// TIA Portal V18 program export: 3 tag tables, 18 data types, 3 data blocks, 44 code blocks (in call order from the OBs), 34 instance data blocks

VAR_GLOBAL   // PLC tag table "Assigned IO"
   HPU_In AT %I0.0 : "Starter_HPU_IO_In";
   HPU_Out AT %Q0.0 : "Starter_HPU_IO_Out";
   Console_In AT %I200.0 : "Console_IO_In";
   Console_Out AT %Q200.0 : "Console_IO_Out";
   ComFault AT %M20.1 : Bool;
   SystemFault AT %M1.0 : Bool;
   RemConsole_In AT %I500.0 : "RemConsole_IO_In";
   RemConsole_Out AT %Q500.0 : "RemConsole_IO_Out";
   RemConEn AT %M29.6 : Bool;   // Remote console is enable if Aux or TD En and heartbeat is ok
END_VAR

VAR_GLOBAL   // PLC tag table "Default tag table"
   TestByte AT %MB2500 : Byte;
   RotaryRPMHMI AT %MD534 : Real;   // It is a absolute value, to display on HMI gauge
   PSIcheck AT %MD544 : Real;
   RotaryStopped AT %M568.0 : Bool;
   MUTorqSetKFtLbs AT %MD570 : Real;
   DrillTorqSetKFtLbs AT %MD574 : Real;
END_VAR
VAR_GLOBAL CONSTANT   // user constants
   RigNumber : Real := 0.0;
   "Program Version" : Real := 0.0;
   RotaryEncInvDir : Bool := 0;   // Used to invert the counting of the rotary encoder
END_VAR

VAR_GLOBAL   // PLC tag table "System Variables"
   RotaryCounts AT %MD100 : DInt;   // Actually rotary count feedback
   RotaryRPM AT %MD104 : Real;   // frequency of rotray feedack
   AuxPumpRunning AT %M10.0 : Bool;   // Status of Aux Pump. 1 Running 0 stopped
   EngineRPMCounts AT %MD108 : DInt;   // CAT Engine RPM count return
   EngineRPMFreq AT %MD112 : Real;   // CAT Engine RPM freqency measured
   CoolingFanRunning AT %M10.1 : Bool;   // Status of Cooler Running 0 stopped
   M1Running AT %M10.2 : Bool;   // Status of P1 Running 0 stopped
   M2Running AT %M10.3 : Bool;   // Status of P2 Running 0 stopped
   AuxPumpHOA AT %M10.4 : Bool;   // Actual Signal to Soft Starter
   CoolingFanHOA AT %M10.5 : Bool;   // Actual Signal to Soft Starter
   M1HOA AT %M10.6 : Bool;   // Actual Signal to Soft Starter
   M2HOA AT %M10.7 : Bool;   // Actual Signal to Soft Starter
   ChargePump1PSw AT %M11.0 : Bool;   // Close = Pressure
   TDLubeFlowSw AT %M11.1 : Bool;   // Close = Flow
   TankLowLevelSw AT %M11.2 : Bool;   // Low Level = Open
   TankHighTempSw AT %M11.3 : Bool;   // High Temp = Open
   TDFwdFilter2 AT %M11.5 : Bool;   // Plugged = Open
   TDRevFilter1 AT %M11.6 : Bool;   // Plugged = Open
   TDRevFilter2 AT %M11.7 : Bool;   // Plugged = Open
   AuxReturnFilter AT %M12.0 : Bool;   // Plugged = Open
   KLoopFilter AT %M12.1 : Bool;   // Plugged = Open
   ChargeFilter AT %M12.2 : Bool;   // Plugged = Open
   M1CurrentRaw AT %MW122 : Int;
   M2CurrentRaw AT %MW128 : Int;
   M1CurrentV AT %MD124 : Real;
   M2CurrentV AT %MD130 : Real;
   TDPressFWDRaw AT %MW134 : Int;   // TD Forward Pressure Input
   TDPressREVRaw AT %MW136 : Int;   // TD Reverse Pressure Input
   ClosedLoopTempRaw AT %MW138 : Int;
   ChargeFlowRaw AT %MW140 : Int;
   HotOilShuttleFlowRaw AT %MW142 : Int;
   AuxFlowRaw AT %MW144 : Int;
   ChargePress1Raw AT %MW146 : Int;
   ChargePress2Raw AT %MW148 : Int;
   TDPressFWDmA AT %MD150 : Real;   // TD Forward Pressure Input
   TDPressREVmA AT %MD154 : Real;   // TD Reverse Pressure Input
   ClosedLoopTempmA AT %MD158 : Real;
   ChargeFlowmA AT %MD162 : Real;
   HotOilShuttleFlowmA AT %MD166 : Real;
   AuxFlowmA AT %MD170 : Real;
   ChargePress1mA AT %MD174 : Real;
   ChargePress2mA AT %MD178 : Real;
   TDP1FwdCmdActRaw AT %MW182 : Int;   // Actual measured output to valve from module
   TDP1RevCmdActRaw AT %MW184 : Int;   // Actual measured output to valve from module
   TDP2FwdCmdActRaw AT %MW186 : Int;   // Actual measured output to valve from module
   TDP2RevCmdActRaw AT %MW188 : Int;   // Actual measured output to valve from module
   TDTorqCmdActRaw AT %MW190 : Int;   // Raw Output to card
   TDP1FwdCmdActmA AT %MD192 : Real;   // Actual measured output to valve from module
   TDP1RevCmdActmA AT %MD196 : Real;   // Actual measured output to valve from module
   TDP2FwdCmdActmA AT %MD200 : Real;   // Actual measured output to valve from module
   TDP2RevCmdActmA AT %MD204 : Real;   // Actual measured output to valve from module
   TDTorqCmdActmA AT %MD208 : Real;   // Actual measured output to valve from module
   LinkRetSw AT %M12.4 : Bool;   // Console Input
   TDAuxSw AT %M12.5 : Bool;   // Console Input
   LinkExtSw AT %M12.6 : Bool;   // Console Input
   TDEnSW AT %M12.7 : Bool;   // Console Input
   HSLT_Sw AT %M13.0 : Bool;   // Console Input
   HandlerFwdSw AT %M13.1 : Bool;   // Console Input
   HandlerRevSw AT %M13.2 : Bool;   // Console Input
   MPNotRunning AT %M13.3 : Bool;   // 0 Pump Running, 1 Pump Not Running - Allowed to Run. Power to permit
   QuillLockSw AT %M13.4 : Bool;   // Console Input
   BUWClSw AT %M13.5 : Bool;   // Console Input
   BUWDnSw AT %M13.6 : Bool;   // Console Input
   BUWUpSw AT %M13.7 : Bool;   // Console Input
   TDModeMUSpinSw AT %M14.0 : Bool;   // Console Input
   TDModeMUTorqSw AT %M14.1 : Bool;   // Console Input
   TDModeDrillRevSw AT %M14.2 : Bool;   // Console Input
   TDModeBreakOutSw AT %M14.3 : Bool;   // Console Input
   ElevOpSw AT %M14.4 : Bool;   // Console Input
   TDExtSw AT %M14.5 : Bool;   // Console Input
   ElevClSw AT %M14.6 : Bool;   // Console Input
   TDRetSw AT %M14.7 : Bool;   // Console Input
   PTO_Sw AT %M15.0 : Bool;   // Console Input
   PurgePressureSw AT %M15.1 : Bool;   // Console Input
   MSVClSw AT %M15.2 : Bool;   // Console Input
   MSVAutoSw AT %M15.3 : Bool;   // Console Input
   MSVOpSw AT %M15.4 : Bool;   // Console Input
   LinkFloatSw AT %M15.5 : Bool;   // Console Input
   MUTorqPotRaw AT %MW212 : Int;
   DrillTorqPotRaw AT %MW214 : Int;
   DrillThrottlePotRaw AT %MW216 : Int;
   MUTorqPotV AT %MD218 : Real;
   DrillTorqPotV AT %MD222 : Real;
   DrillThrottlePotV AT %MD226 : Real;
   RotEncLDSlot AT %MB230 : Byte;   // Bit 0-3 Slot 0, Bit 4-7 Slot 1. 0 0 0 0 for Idle, 0 0 0 1 Load Counter
   TDFwdPress1Raw AT %MD240 : UDInt;   // Pump 1 Forward Pressure output
   TDFwdPress2Raw AT %MD244 : UDInt;   // Pump 2 Forward Pressure output
   TDRevPress1Raw AT %MD248 : UDInt;   // Pump 1 Rev Pressure output
   TDRevPress2Raw AT %MD252 : UDInt;   // Pump 2 Rev Pressure output
   TDTorqPressRaw AT %MD256 : UDInt;   // Torq Output
   TDFwdPress1En AT %M15.6 : Bool;   // Enable Pump 1 Forward Pressure output
   TDFwdPress2En AT %M15.7 : Bool;   // Enable Pump 2 Forward Pressure output
   TDRevPress1En AT %M16.0 : Bool;   // Enable Pump 1 Rev Pressure output
   TDRevPress2En AT %M16.1 : Bool;   // Enable Pump 2 Rev Pressure output
   TDTorqPressEn AT %M16.2 : Bool;   // Enable Torq output
   BUWClSol AT %M16.4 : Bool;
   HSLT_Sol AT %M16.5 : Bool;
   ElevClSol AT %M16.6 : Bool;
   ElevOpSol AT %M16.7 : Bool;
   LinkExtSol AT %M17.0 : Bool;
   LinkRetSol AT %M17.1 : Bool;
   LinkFloatSol AT %M17.2 : Bool;
   LSHT_Sol AT %M17.3 : Bool;
   MSVOpSol AT %M17.4 : Bool;
   MSVClSol AT %M17.5 : Bool;
   BUWDnSol AT %M17.6 : Bool;
   BUWUpSol AT %M17.7 : Bool;
   HandlerFWDSol AT %M18.0 : Bool;
   HandlerREVSol AT %M18.1 : Bool;
   TDExtSol AT %M18.2 : Bool;
   TDRetSol AT %M18.3 : Bool;   // Output Coil
   HourMeterOn AT %M18.4 : Bool;
   EngRampSpeedDn AT %M18.5 : Bool;
   AuxPumpStart AT %M18.6 : Bool;
   EngRampSpeedUp AT %M18.7 : Bool;
   CoolingFanStart AT %M19.0 : Bool;
   FailSafeEnSol AT %M19.1 : Bool;
   PumpEnSol AT %M19.2 : Bool;   // CAT/Rig 11 Only
   BOControlSol AT %M19.3 : Bool;
   AuxUnloaderSol AT %M19.4 : Bool;
   HotOilControlSol AT %M19.5 : Bool;
   BUWOpSol AT %M19.6 : Bool;
   BypassValveSol AT %M19.7 : Bool;
   TDFwdPress1mA AT %MD260 : Real;   // Pump 1 Forward Pressure output
   TDFwdPress2mA AT %MD264 : Real;   // Pump 2 Forward Pressure output
   TDRevPress1mA AT %MD268 : Real;   // Pump 1 Rev Pressure output
   TDRevPress2mA AT %MD272 : Real;   // Pump 2 Rev Pressure output
   TDTorqPressmA AT %MD276 : Real;   // Torq Output
   PTOLED AT %M20.4 : Bool;
   HPUFaultLED AT %M20.5 : Bool;
   TDFlushFaultLED AT %M20.6 : Bool;
   BUWClLED AT %M20.7 : Bool;
   TDEnLED AT %M21.0 : Bool;
   ConLowPurgeLED AT %M21.1 : Bool;
   MSVClLED AT %M21.2 : Bool;   // Mud Saver valve closed LED
   QuillLockLED AT %M21.3 : Bool;
   ElevClLED AT %M21.4 : Bool;
   Horn AT %M21.5 : Bool;
   MSVClInt AT %M21.6 : Bool;   // Mud saver valve closed interlocks outputs
   BUWClInt AT %M21.7 : Bool;   // BUW Closed interlock outputs
   DrillRecTorqRaw AT %MW280 : Int;
   DrillRecRPMRaw AT %MW282 : Int;
   DrillRecTorqFtLbs AT %MD284 : Real;
   DrillRecRPM AT %MD288 : Real;
   DrillRecTorqmA AT %MD292 : Real;
   DrillRecRPMmA AT %MD296 : Real;
   RotEncUnFl AT %M22.0 : Bool;   // Encoder underflow
   RotEncOvFl AT %M22.1 : Bool;   // Encoder OVerflow
   RotEncPosReset AT %M22.2 : Bool;   // Set high to trigger zero position of encoder. Bit will reset once position reset
   RotEncSlot0 AT %MD232 : Real;
   RotEncSlot1 AT %MD236 : Real;
   TDRotStopped AT %M22.3 : Bool;   // Set if TD has not moved after stop time elapsed
   RotAbsPosDeg AT %MD300 : Real;   // Absolute rotary position from zero point
   RotRelPosDeg AT %MD304 : Real;   // Position from 0-360 degrees
   RotPosTurns AT %MD308 : Real;   // Turns from zero point
   TDFlushFlowSw AT %M22.4 : Bool;
   M1Current AT %MD312 : Real;
   M2Current AT %MD316 : Real;
   TDPressFwdPSI AT %MD320 : Real;   // TD Fwd Pressure PSI
   TDPressRevPSI AT %MD324 : Real;   // TD Rev Pressure PSI
   ClosedLoopTempC AT %MD328 : Real;   // Closed Loop Temp in C
   ChargeFlowGPM AT %MD332 : Real;   // Charge Flow in GPM
   HotOilFlowGPM AT %MD336 : Real;   // Hot Oil Shuttle Flow in GPM
   AuxFlowGPM AT %MD340 : Real;   // Aux Flow GPM
   ChargePress1PSI AT %MD344 : Real;   // Charge Pump 1 Pressure PSI
   ChargePress2PSI AT %MD348 : Real;   // Charge Pump 2 Pressure PSI
   M1CurrentFilt AT %MD352 : Real;
   M2CurrentFilt AT %MD356 : Real;
   TDPressFwdPSIFilt AT %MD360 : Real;
   TDPressRevPSIFilt AT %MD364 : Real;
   ClosedLoopTempCFilt AT %MD368 : Real;
   ChargeFlowGPMFilt AT %MD372 : Real;
   HotOilFlowGPMFilt AT %MD376 : Real;
   AuxFlowGPMFilt AT %MD380 : Real;
   ChargePress1PSIFilt AT %MD384 : Real;
   ChargePress2PSIFilt AT %MD388 : Real;
   AuxPumpHand AT %M22.5 : Bool;   // Starter HOA switch in the Hand Position
   AuxPumpOff AT %M22.6 : Bool;   // Starter HOA switch in the Off position
   CoolingFanHand AT %M23.0 : Bool;   // Starter HOA switch in the Hand Position
   CoolingFanOff AT %M23.1 : Bool;   // Starter HOA switch in the Off position
   M1Hand AT %M23.3 : Bool;   // Starter HOA switch in the Hand Position
   M1Off AT %M23.4 : Bool;   // Starter HOA switch in the Off position
   M2Hand AT %M23.6 : Bool;   // Starter HOA switch in the Hand Position
   M2Off AT %M23.7 : Bool;   // Starter HOA switch in the Off position
   AuxPumpFault AT %M22.7 : Bool;   // Motor failed to start before motor timeout time
   CoolingFanFault AT %M23.2 : Bool;   // Motor failed to start before motor timeout time
   M1Fault AT %M23.5 : Bool;   // Motor failed to start before motor timeout time
   M2Fault AT %M24.0 : Bool;   // Motor failed to start before motor timeout time
   M1Start AT %M20.2 : Bool;   // Start Motor 1
   M2Start AT %M20.3 : Bool;   // Start Motor 2
   BypassStart AT %M24.1 : Bool;   // Ready for Bypass to start, waiting for PTO
   BypassRunning AT %M24.2 : Bool;   // Latched Signal set if PTO pressed after Bypass Start
   StartCAT AT %M24.3 : Bool;   // Indicates CAT startup up. System ramps up and will enable.
   BUWMaintConfirm AT %M24.4 : Bool;
   PTOConfirmed AT %M24.5 : Bool;   // PTO Confirm pulse for 5 seconds after button pressed
   BUWOpenClk AT %M24.6 : Bool;   // Periodic clock signal that will be on for 5 seconds and off for 1 min. Used for maintain gripper open
   BUWAutoCl AT %M24.7 : Bool;   // Latch for Gripper Close
   BUWAutoClHold AT %M25.0 : Bool;   // LAtch for Gripper Hold Closed
   BUWAutoOp AT %M25.1 : Bool;   // Lath for Gripper Open
   OscSpeedfwdHold AT %M25.2 : Bool;
   QuillLockEnabled AT %M25.3 : Bool;   // Bit used to know if Quill Lock allowed
   BUWClHoldTime AT %M25.4 : Bool;   // On for half a second to hold the close before turning off
   MUTorqPotPer AT %MD392 : Real;
   DrillTorqPotPer AT %MD396 : Real;
   DrillThrottlePotPer AT %MD400 : Real;
   MUTorqPotPerFilt AT %MD404 : Real;
   DrillTorqPotPerFilt AT %MD408 : Real;
   DrillThrottlePotPerFilt AT %MD412 : Real;
   ActTorqFtLbs AT %MD416 : Real;   // Calculated actual torque
   ActTorqFtLbsFilt AT %MD420 : Real;   // Filtered Actual Torque
   TDDifPressPSI AT %MD424 : Real;   // Diffential pressure betweeen FWD and REV
   DrillTorqSetFtLbs AT %MD428 : Real;   // Internal setpoint value from the console input FtLbs
   MUTorqSetFtLbs AT %MD432 : Real;   // Internal setpoint value from the console input FtLbs
   RotDegPerCount AT %MD436 : Real;   // Actual Degrees per Count for current encoder setup
   DrillTorqSetMax AT %MD440 : Real;   // Maximum value allowed to set drill torq too based on MU torq settings
   BOCycleDone AT %M25.6 : Bool;   // Trigger when BO Sw released
   MUCycleDone AT %M25.7 : Bool;   // Set when MU done
   MUSwRelease AT %M26.0 : Bool;   // Trigger when MU SW released
   MUDoneSetFtLbs AT %MD444 : Real;   // Minimum torque to surpass to declare MU Done
   ElevClFeedback AT %M12.3 : Bool;   // Feedback switch that the elevators are closed
   LamptTest AT %M26.1 : Bool;   // Bit Used to trigger Lamp to turn on.
   FlushFaultNoSpin AT %M26.2 : Bool;   // TD flush faulted. No Spin allowed
   ThrottleDisable AT %M26.3 : Bool;   // Throttle disable if high
   ThrottleUnlocked AT %M26.4 : Bool;   // Throttle boots up locked. Must be below zero to enable after startup
   DrillTorqLimited AT %M26.5 : Bool;   // Set high if max drill torq limited by max makeup torq
   DrillTorqSetPSI AT %MD448 : Real;   // PSI equivalent to get desired torq from valve
   MUTorqSetPSI AT %MD452 : Real;   // PSI equivalent to get desired torq from valve
   TDStart AT %M25.5 : Bool;   // Bit will be set High when TD is started for regular operations
   BypassPTO AT %M26.6 : Bool;   // Bypass PTO accept
   BypassOutEnable AT %M26.7 : Bool;   // Bypass control enabled to allow signal to Pumps after delay
   BypassHighTemp AT %M27.0 : Bool;   // High Closed loop temp in bypass mode
   TDPressTxFault AT %M27.1 : Bool;   // One of the pressure transducers if not working. No auto MU
   HSLTDisThrottle AT %M27.2 : Bool;   // Bit high after shift to disable throttle
   LSHTDisThrottle AT %M27.3 : Bool;   // Bit high after shift to disable throttle
   MUSeqRunning AT %M27.4 : Bool;   // Bool indicating mak up sequence is running.
   AutoMUTorqLow AT %M27.5 : Bool;   // Auto Make Up Low Torque range
   AutoMUTorqMid AT %M27.6 : Bool;   // Auto Make Up Mid Torque Range
   AutoMuTorqHigh AT %M27.7 : Bool;   // Auto Make Up High Torque Range
   HiTempRPMRed AT %M28.1 : Bool;   // Bit indicating high temperature and RPM to be reduced
   HiTempShutdown AT %M28.2 : Bool;   // Bit indicating high temperature and shutdown needed.
   TDRotDirFwd AT %M28.3 : Bool;   // Rotary moving fwd
   TDRotDirRev AT %M28.4 : Bool;   // Rotary moving rev
   ActTorqKFtLbsFilt AT %MD456 : Real;
   RotEncA AT %M28.5 : Bool;
   RotEncB AT %M28.6 : Bool;
   BOSeqRunning AT %M28.0 : Bool;   // Bool indicating break out sequence is running.   {ExternalVisible false}
   HPU_AiV2SpareRaw AT %MW460 : Int;   // Spare Analog Voltage Input Raw
   HPU_AiV2SpareV AT %MD472 : Real;   // Spare Analog Voltage Input
   HPU_AiV3SpareRaw AT %MW462 : Int;   // Spare Analog Voltage Input Raw
   HPU_AiV4SpareRaw AT %MW464 : Int;   // Spare Analog Voltage Input Raw
   HPU_AiV5SpareRaw AT %MW466 : Int;   // Spare Analog Voltage Input Raw
   HPU_AiV6SpareRaw AT %MW468 : Int;   // Spare Analog Voltage Input Raw
   HPU_AiV7SpareRaw AT %MW470 : Int;   // Spare Analog Voltage Input Raw
   HPU_AiV3SpareV AT %MD476 : Real;   // Spare Analog Voltage Input
   HPU_AiV4SpareV AT %MD480 : Real;   // Spare Analog Voltage Input
   HPU_AiV5SpareV AT %MD484 : Real;   // Spare Analog Voltage Input
   HPU_AiV6SpareV AT %MD488 : Real;   // Spare Analog Voltage Input
   HPU_AiV7SpareV AT %MD492 : Real;   // Spare Analog Voltage Input
   Con_AiV3SpareRaw AT %MW496 : Int;   // Spare Analog Voltage Input Raw
   Con_AiV4SpareRaw AT %MW498 : Int;   // Spare Analog Voltage Input Raw
   Con_AiV5SpareRaw AT %MW500 : Int;   // Spare Analog Voltage Input Raw
   Con_AiV6SpareRaw AT %MW502 : Int;   // Spare Analog Voltage Input Raw
   Con_AiV7SpareRaw AT %MW504 : Int;   // Spare Analog Voltage Input Raw
   Con_AiV3SpareV AT %MD506 : Real;   // Spare Analog Voltage Input
   Con_AiV4SpareV AT %MD510 : Real;   // Spare Analog Voltage Input
   Con_AiV5SpareV AT %MD514 : Real;   // Spare Analog Voltage Input
   Con_AiV6SpareV AT %MD518 : Real;   // Spare Analog Voltage Input
   Con_AiV7SpareV AT %MD522 : Real;   // Spare Analog Voltage Input
   HornTest AT %M28.7 : Bool;
   Charge1Fault AT %M29.0 : Bool;   // Charge pressure fault while TD enabled
   FilterPlugged AT %M29.1 : Bool;
   Clock_Byte AT %MB0 : Byte;
   Clock_10Hz AT %M0.0 : Bool;   // 0.1 s period
   Clock_5Hz AT %M0.1 : Bool;   // 0.2 s period
   "Clock_2.5Hz" AT %M0.2 : Bool;   // 0.4 s period
   Clock_2Hz AT %M0.3 : Bool;   // .06 s period
   "Clock_1.25Hz" AT %M0.4 : Bool;   // 0.8s period
   Clock_1Hz AT %M0.5 : Bool;   // 1s period
   "Clock_0.625Hz" AT %M0.6 : Bool;   // 1.6s period
   "Clock_0.5Hz" AT %M0.7 : Bool;   // 2.0 s period
   HiTempAlarm AT %M29.2 : Bool;
   LubeFlowFault AT %M29.3 : Bool;
   HornSilence AT %M29.4 : Bool;
   EngineFault AT %M29.5 : Bool;   // CAT Engine Fault. Below min RPM
   EngineRPM AT %MD116 : Real;
   ClosedLoopTempCMax AT %MD526 : Real;
   TDEnabled AT %M16.3 : Bool;   // Start Request received and system enabled
   Charge2Fault AT %M20.0 : Bool;
   ChargePump2PSw AT %M29.7 : Bool;   // Close = Pressure
   TDFwdFilter1 AT %M11.4 : Bool;   // Plugged = Open
   LastCount AT %MD30 : DInt;
   RotRelPosDegHMIPos AT %MD34 : Real;
   OscHomeRelDegHMIPos AT %MD530 : Real;
   SwitchSWGATE AT %M538.0 : Bool;
   OscSpeedrevHold AT %M38.0 : Bool;
   RevFwdPause AT %M38.1 : Bool;
   FwdRevPasue AT %M38.2 : Bool;
   PSIadjustbit AT %M38.3 : Bool;
   PSIdrillTorquCalca AT %MD540 : Real;
   PSIsettle AT %MD548 : Real;
   PSIadjustRange AT %MD552 : Real;
   PSIadjustval AT %MD556 : Real;
   ClosedLoopTempF AT %MD560 : Real;
   RotaryRPMActual AT %MD564 : Real;
END_VAR
VAR_GLOBAL CONSTANT   // user constants
   AlwaysOn : Bool := 1;
   AlwaysOff : Bool := 0;
END_VAR

TYPE "Console_IO_In"
   STRUCT
      Slot1 { S7_SetPoint := 'True'} : "DI16x24V_In";
      Slot2 { S7_SetPoint := 'True'} : "DI16x24V_In";
      Slot3 { S7_SetPoint := 'True'} : "AI8xU_In";
   END_STRUCT;
END_TYPE

TYPE "Console_IO_Out"
   STRUCT
      Slot4 : "DQ16x24V_Out";
      Slot5 : "AQ4xI/U_Out";
   END_STRUCT;
END_TYPE

TYPE "RemConsole_IO_In"
   STRUCT
      Element_1 : Bool;
      Element_2 : Bool;
      Element_3 : Bool;
      Element_4 : Bool;
      Element_5 : Bool;
      Element_6 : Bool;
      Element_7 : Bool;
      LinkTiltRetr : Bool;
      TopDriveAux : Bool;
      LinkTiltExt : Bool;
      TopDriveEn : Bool;
      HSLTEn : Bool;
      HandlerFwd : Bool;
      HandlerRev : Bool;
      MudPumpRunning : Bool;
      QuillLock : Bool;
      BUWClose : Bool;
      BUWDown : Bool;
      BUWUp : Bool;
      TDModeMUSpin : Bool;
      TDModeMUTorq : Bool;
      TDModeRev : Bool;
      TDModeBO : Bool;
      ElevOp : Bool;
      TDExt : Bool;
      ElevCl : Bool;
      TDRet : Bool;
      PTO : Bool;
      Spare : Bool;
      MSVClose : Bool;
      MSVAuto : Bool;
      MSVOpen : Bool;
      LinkTiltFloat : Bool;
      Spare_1 : Bool;
      Spare_2 : Bool;
      Spare_3 : Bool;
      Spare_4 : Bool;
      Spare_5 : Bool;
      Heartbeat : Bool;
      Reserved : Byte;
      MUTorqLim : Int;
      DrillTorqLim : Int;
      DrillThrottle : Int;
      SpareAI : Int;
      SpareAI_1 : Int;
      SpareAI_2 : Int;
      SpareAI_3 : Int;
      SpareAI_1_1 : Int;
   END_STRUCT;
END_TYPE

TYPE "RemConsole_IO_Out"
   STRUCT
      PTOLED : Bool;
      HPUFaultLED : Bool;
      TDFaultLED : Bool;
      BUWClLED : Bool;
      TDEnLED : Bool;
      Spare_6 : Bool;
      MSVClLED : Bool;
      QuillLockedLED : Bool;
      ElevClLED : Bool;
      Horn : Bool;
      MSVClInt : Bool;
      BUWClInt : Bool;
      Spare_7 : Bool;
      Spare_8 : Bool;
      Spare_9 : Bool;
      Spare_10 : Bool;
      Spare_11 : Bool;
      Spare_12 : Bool;
      Spare_13 : Bool;
      Spare_14 : Bool;
      Spare_15 : Bool;
      Spare : Bool;
      Spare_16 : Bool;
      Spare_17 : Bool;
      Spare_18 : Bool;
      Spare_19 : Bool;
      Spare_1 : Bool;
      Spare_2 : Bool;
      Spare_3 : Bool;
      Spare_4 : Bool;
      Spare_5 : Bool;
      Spare_20 : Bool;
      DrillRecTorq : Int;
      DrillRecRPM : Int;
      SpareAO : Int;
      SpareAO_2 : Int;
   END_STRUCT;
END_TYPE

TYPE "Runtime_Out"
   STRUCT
      TotalTime : DInt;
      TotHours : DInt;
      TotMins : DInt;
      TotSeconds : DInt;
      CurrentTime : DInt;   // Current Time in Seconds
      CurHours : DInt;
      CurMins : DInt;
      CurSeconds : DInt;
   END_STRUCT;
END_TYPE

TYPE "Starter_HPU_IO_In"
   STRUCT
      Slot2 { ExternalWritable := 'False'} : "TM_Count_Man_In";
      Slot3 { ExternalWritable := 'False'} : "DI16x24V_In";
      Slot4 { ExternalWritable := 'False'} : "DI16x24V_In";
      Slot5 { S7_SetPoint := 'True'} : "AI8xU_In";
      Slot6 { ExternalWritable := 'False'} : "AI8xI_In";
      Slot7 { ExternalWritable := 'False'} : "TM_Pulse_2x24_In";
      Slot8 { S7_SetPoint := 'True'} : "TM_Pulse_2x24_In";
      Slot9 { S7_SetPoint := 'True'} : "TM_Pulse_2x24_In";
   END_STRUCT;
END_TYPE

TYPE "Starter_HPU_IO_Out"
   STRUCT
      Slot2 { S7_SetPoint := 'True'} : "TM_Count_Man_Out";
      Slot7 { S7_SetPoint := 'True'} : "TM_Pulse_2x24_Out";
      Slot8 { S7_SetPoint := 'True'} : "TM_Pulse_2x24_Out";
      Slot9 { S7_SetPoint := 'True'} : "TM_Pulse_2x24_Out";
      Slot10 { S7_SetPoint := 'True'} : "RQ_4x120VDC/5A_In";
      Slot11 { S7_SetPoint := 'True'} : "RQ_4x120VDC/5A_In";
      Slot12 { S7_SetPoint := 'True'} : "RQ_4x120VDC/5A_In";
      Slot13 { S7_SetPoint := 'True'} : "RQ_4x120VDC/5A_In";
      Slot14 { S7_SetPoint := 'True'} : "RQ_4x120VDC/5A_In";
      Slot15 { S7_SetPoint := 'True'} : "RQ_4x120VDC/5A_In";
      Slot16 { S7_SetPoint := 'True'} : "RQ_4x120VDC/5A_In";
      Slot17 { S7_SetPoint := 'True'} : "RQ_4x120VDC/5A_In";
   END_STRUCT;
END_TYPE

TYPE "TD_Modes"
   STRUCT
      Drill : Int;
      DrillReverse : Int := 1;
      MUSpin : Int := 2;
      MUTorque : Int := 3;
      BO : Int := 4;
      Oscillate : Int := 5;
      Bypass : Int := 6;
   END_STRUCT;
END_TYPE

TYPE "AI8xI_In"
   STRUCT
      Ch0 : Int;
      Ch1 : Int;
      Ch2 : Int;
      Ch3 : Int;
      Ch4 : Int;
      Ch5 : Int;
      Ch6 : Int;
      Ch7 : Int;
   END_STRUCT;
END_TYPE

TYPE "AI8xU_In"
   STRUCT
      Ch0 : Int;
      Ch1 : Int;
      Ch2 : Int;
      Ch3 : Int;
      Ch4 : Int;
      Ch5 : Int;
      Ch6 : Int;
      Ch7 : Int;
   END_STRUCT;
END_TYPE

TYPE "DI16x24V_In"
   STRUCT
      Ch0 : Bool;
      Ch1 : Bool;
      Ch2 : Bool;
      Ch3 : Bool;
      Ch4 : Bool;
      Ch5 : Bool;
      Ch6 : Bool;
      Ch7 : Bool;
      Ch8 : Bool;
      Ch9 : Bool;
      Ch10 : Bool;
      Ch11 : Bool;
      Ch12 : Bool;
      Ch13 : Bool;
      Ch14 : Bool;
      Ch15 : Bool;
   END_STRUCT;
END_TYPE

TYPE "DQ16x24V_Out"
   STRUCT
      Ch0 : Bool;
      Ch1 : Bool;
      Ch2 : Bool;
      Ch3 : Bool;
      Ch4 : Bool;
      Ch5 : Bool;
      Ch6 : Bool;
      Ch7 : Bool;
      Ch8 : Bool;
      Ch9 : Bool;
      Ch10 : Bool;
      Ch11 : Bool;
      Ch12 : Bool;
      Ch13 : Bool;
      Ch14 : Bool;
      Ch15 : Bool;
   END_STRUCT;
END_TYPE

TYPE "TM_Count_Man_In"
   STRUCT
      COUNT_VALUE : DInt;
      CAPTURED_VALUE : DInt;
      MEASURED_VALUE : DInt;
      POWER_ERROR : Bool;
      ENC_ERROR : Bool;
      LD_ERROR : Bool;
      Reserved1 : Bool;
      Reserved2 : Bool;
      Reserved3 : Bool;
      Reserved4 : Bool;
      Reserved5 : Bool;
      Reserved6 : Bool;
      RES_EVENT_ACK : Bool;
      LD_STS_SLOT0 : Bool;
      LD_STS_SLOT1 : Bool;
      STS_READY : Bool;
      STS_SW_GATE : Bool;
      Reserved7 : Bool;
      Reserved8 : Bool;
      STS_DIR : Bool;
      STS_CNT : Bool;
      STS_GATE : Bool;
      STS_DQ0 : Bool;
      STS_DQ1 : Bool;
      STS_DI0 : Bool;
      STS_DI1 : Bool;
      STS_DI2 : Bool;
      EVENT_ZERO : Bool;
      EVENT_UFLW : Bool;
      EVENT_OFLW : Bool;
      EVENT_CMP0 : Bool;
      EVENT_CMP1 : Bool;
      EVENT_SYNC : Bool;
      EVENT_CAP : Bool;
      STS_M_INTERVAL : Bool;
   END_STRUCT;
END_TYPE

TYPE "TM_Count_Man_Out"
   STRUCT
      SLOT_0 : Real;
      SLOT_1 : Real;
      LD_SLOT_0_1 : Byte;
      SW_GATE : Bool;
      TM_CTRL_DQ0 : Bool;
      TM_CTRL_DQ1 : Bool;
      SET_DQ0 : Bool;
      SET_DQ1 : Bool;
      EN_SYNC_UP : Bool;
      EN_SYNC_DN : Bool;
      EN_CAPTURE : Bool;
      RES_ERROR : Bool;
      RES_EVENT : Bool;
      Reserved1 : Bool;
      Reserved2 : Bool;
      Reserved3 : Bool;
      Reserved4 : Bool;
      Reserved5 : Bool;
      SET_DIR : Bool;
      Reserved : Byte;
   END_STRUCT;
END_TYPE

TYPE "TM_Pulse_2x24_In"
   STRUCT
      Ch0 { S7_SetPoint := 'True'} : "TM_Pulse_2x24_In_PWM";
      Ch1 { S7_SetPoint := 'True'} : "TM_Pulse_2x24_In_PWM";
   END_STRUCT;
END_TYPE

TYPE "TM_Pulse_2x24_In_PWM"
   STRUCT
      ERR_PWR : Bool;
      ERR_24V : Bool;
      ERR_LD : Bool;
      Reserved5 : Bool;
      ERR_DQA : Bool;
      ERR_DQB : Bool;
      ERR_OUT_VAL : Bool;
      ERR_SLOT_VAL : Bool;
      Reserved0 : Bool;
      Reserved1 : Bool;
      STS_LD_SLOT : Bool;
      Reserved2 : Bool;
      STS_READY : Bool;
      STS_SW_ENABLE : Bool;
      Reserved3 : Bool;
      Reserved4 : Bool;
      STS_ENABLE : Bool;
      STS_DQA : Bool;
      STS_DQB : Bool;
      STS_DI : Bool;
      STS_DITHER : Bool;
      Reserved6 : Bool;
      Reserved7 : Bool;
      Reserved8 : Bool;
      MEASURE_CURRENT : Int;
      QLMN_LLM : Bool;
      QLMN_HLM : Bool;
      Reserved9 : Bool;
      Reserved10 : Bool;
      Reserved11 : Bool;
      Reserved12 : Bool;
      Reserved13 : Bool;
      Reserved14 : Bool;
      Reserved15 : Byte;
   END_STRUCT;
END_TYPE

TYPE "TM_Pulse_2x24_Out"
   STRUCT
      Ch0 : "TM_Pulse_2x24_Out_PWM";
      Ch1 { S7_SetPoint := 'True'} : "TM_Pulse_2x24_Out_PWM";
   END_STRUCT;
END_TYPE

TYPE "TM_Pulse_2x24_Out_PWM"
   STRUCT
      OUTPUT_VALUE : UDInt;   // Pulse Duration
      SLOT : UDInt;   // Load Value
      LD_SLOT_Bit0 : Bool;
      LD_SLOT_Bit1 : Bool;
      LD_SLOT_Bit2 : Bool;
      LD_SLOT_Bit3 : Bool;
      MODE_SLOT : Bool;
      Reserved1 : Bool;
      Reserved2 : Bool;
      Reserved3 : Bool;
      SW_ENABLE : Bool;
      TM_CTRL_DQ : Bool;
      Reserved4 : Bool;
      SET_DQA : Bool;
      SET_DQB : Bool;
      DITHER : Bool;
      Rerserved6 : Bool;
      Rerserved7 : Bool;
      RES_ERROR : Bool;
      Reserved8 : Bool;
      Reserved9 : Bool;
      Reserved10 : Bool;
      Reserved11 : Bool;
      Reserved12 : Bool;
      Reserved13 : Bool;
      Reserved14 : Bool;
      Rerserved : Byte;
   END_STRUCT;
END_TYPE

DATA_BLOCK "CoordinationHmi"   // DB1
{ S7_Optimized_Access := 'FALSE' }
// stored: AutoNumber false
   VAR
      CoordinationConsoleHmi : Array[0..15] of Bool;
      CoordinationHpuHmi : Array[0..15] of Bool;
      CoordinationDoghouseHmi : Array[0..15] of Bool;
      RTClock : DTL;
   END_VAR
BEGIN
END_DATA_BLOCK

DATA_BLOCK "IO_Settings"   // DB101
{ S7_Optimized_Access := 'TRUE' }
// This datablock will hold the IO setup settings for the unit
// stored: AutoNumber false, MemoryReserve 100
   VAR RETAIN
      ChargePress1Tx { S7_SetPoint := 'True'} : Bool;   // Charge Pressure Transducer Exist - used for alarms
      ChargePress1Sw { S7_SetPoint := 'True'} : Bool;
      ChargePress2Tx { S7_SetPoint := 'True'} : Bool;   // Charge Pressure Transducer Exist - used for alarms
      ChargePress2Sw { S7_SetPoint := 'True'} : Bool;
      SecondaryFilters { S7_SetPoint := 'True'} : Bool;   // Set bit if 2 FWD and REV filters exist.
      HPUType { S7_SetPoint := 'True'} : Int;   // 0 = Elec HPU , 1 = CAT HPU
      LubeFlowSwitch { S7_SetPoint := 'True'} : Bool;   // Set if TD is equiped with Lube Flow Switch
      KLoopFilter { S7_SetPoint := 'True'} : Bool;   // Set if KL Filter is equipped
      ElevClSw { S7_SetPoint := 'True'} : Bool;   // Set if Elevator Close Switch exists
   END_VAR
BEGIN
END_DATA_BLOCK

DATA_BLOCK "Settings"   // DB100
{ S7_Optimized_Access := 'TRUE' }
// stored: AutoNumber false, MemoryReserve 100
   VAR RETAIN
      ActTorqAlpha { S7_SetPoint := 'True'} : Real := 0.0;   // Low Pass Filter, Alpha be >= 0 and < 1. 0 No filterting.
      AlarmDebounce { S7_SetPoint := 'True'} : Time := T#500MS;   // Time an alarm must be present before setting
      MUTorqAutoSet1per { S7_SetPoint := 'True'} : Real := 65.0;   // Perfent of MU a torq low Set point to allow full speed ramp
      MUTorqAutoSet2per { S7_SetPoint := 'True'} : Real := 90.0;   // Percent of MU Torq high setpoint to say complete
      MUAutoHoldTime { S7_SetPoint := 'True'} : Time := T#2S_150MS;   // Time System will hold max torq before ramping down
      MUAutoSlewLow { S7_SetPoint := 'True'} : Real := 150.0;   // Slew rate for Auto make up rising in low torque. mA/Sec
      MUAutoSlewMid { S7_SetPoint := 'True'} : Real := 25.0;   // Slew rate for Auto make up rising in mid torq. mA/Sec
      AuxFlowMinGPM { S7_SetPoint := 'True'} : Real := 5.0;   // Min Value of flow transducer
      AuxFlowMaxGPM { S7_SetPoint := 'True'} : Real := 25.0;   // MAx Value of flow transducer
      AuxFlowAlpha { S7_SetPoint := 'True'} : Real := 0.0;   // Low Pass Filter, Alpha be >= 0 and < 1. 0 No filterting.
      BOFlowSlewRise { S7_SetPoint := 'True'} : Real := 500.0;   // Rising Slew Rate mA/sec on Flow Output
      BOFlowSlewFall { S7_SetPoint := 'True'} : Real := 80.0;   // Falling Slew Rate mA/sec on Flow Output
      BOSpinFactor { S7_SetPoint := 'True'} : Real := 1.25;   // BO Flow will be set to MU Spin Percent times this factor to break connection. before slowing back down to Spin Speed
      BOShiftRPM { S7_SetPoint := 'True'} : Real := 4.0;   // In BO above this speed, system will switch from BO Speed setting to Spin setting
      BypassTime { S7_SetPoint := 'True'} : Time := T#2S;   // Time for Bypass to finish running
      BypassFlowPer { S7_SetPoint := 'True'} : Real := 50.0;   // Output to flow in percent valve in Bypass mode
      BypassTorqFtlbs { S7_SetPoint := 'True'} : Real := 12000.0;   // Output to torqur valve in Bypass mode. Actual Value TBD
      CATEngPPR { S7_SetPoint := 'True'} : Int := 113;   // CAT Engine PPR.
      CATMinRPM { S7_SetPoint := 'True'} : Real := 1200.0;   // Minimum running RPM of CAT. Used to trigger Enginer fault
      CATFaultTime { S7_SetPoint := 'True'} : Time := T#15S;   // Time for CAT to get up to speed before fault
      ChargeFlowMinGPM { S7_SetPoint := 'True'} : Real := 5.0;   // Min Value of flow transducer
      ChargeFlowMaxGPM { S7_SetPoint := 'True'} : Real := 1000.0;   // MAx Value of flow transducer
      ChargeFlowAlpha { S7_SetPoint := 'True'} : Real := 0.0;   // Low Pass Filter, Alpha be >= 0 and < 1. 0 No filterting.
      ChargePress1Min { S7_SetPoint := 'True'} : Real := 0.0;   // Min value of transducer range
      ChargePress1Max { S7_SetPoint := 'True'} : Real := 6000.0;   // Max Value of transducer range
      ChargePress1Alpha { S7_SetPoint := 'True'} : Real := 0.0;   // Low Pass Filter, Alpha be >= 0 and < 1. 0 No filterting.
      ChargePress2Min { S7_SetPoint := 'True'} : Real := 0.0;   // Min value of transducer range
      ChargePress2Max { S7_SetPoint := 'True'} : Real := 6000.0;   // Max Value of transducer range
      ChargePress2Alpha { S7_SetPoint := 'True'} : Real := -7111.111;   // Low Pass Filter, Alpha be >= 0 and < 1. 0 No filterting.
      ChargeFaultMinPress { S7_SetPoint := 'True'} : Real := 200.0;   // Min charge pressure before fault shown
      ChargeFaultMaxPress { S7_SetPoint := 'True'} : Real := 1000.0;   // Max Charge pressure before fautl
      CLTempMinC { S7_SetPoint := 'True'} : Real := 0.0;   // Min value of Closed loop Temp transducer
      CLTempMaxC { S7_SetPoint := 'True'} : Real := 204.0;   // Max value of Closed loop Temp transducer
      CLTempMinF { S7_SetPoint := 'True'} : Real := 0.0;
      CLTempMaxF { S7_SetPoint := 'True'} : Real := 400.0;
      CLTempAlpha { S7_SetPoint := 'True'} : Real := 0.0;   // Low Pass Filter, Alpha be >= 0 and < 1. 0 No filterting.
   END_VAR
   VAR
      CLHiTempAlarmF : Real := 158.0;
   END_VAR
   VAR RETAIN
      CLHiTempAlarm { S7_SetPoint := 'True'} : Real := 70.0;   // Closed loop temp in C where alarm comes on. Value for Mobil SCH S26 - Hydrex MV60 - 64
   END_VAR
   VAR
      CLHiTempRPMF : Real := 161.6;
   END_VAR
   VAR RETAIN
      ClHiTempRPM { S7_SetPoint := 'True'} : Real := 72.0;   // Closed loop temp in c where RPM is reduced Value for Mobil SCH S26 - Hydrex MV60 - 66
   END_VAR
   VAR
      ClHiTempShutdownF : Real := 165.2;
   END_VAR
   VAR RETAIN
      ClHiTempShutdown { S7_SetPoint := 'True'} : Real := 74.0;   // Closed loop temp in C where TD shutsdown Value for Mobil SCH S26 - Hydrex MV60 - 68
   END_VAR
   VAR
      ClHiTempBypassF : Real := 161.6;
   END_VAR
   VAR RETAIN
      ClHiTempBypass { S7_SetPoint := 'True'} : Real := 72.0;   // Closed loop Temp in C where Bypass stopped Value for Mobil SCH S26 - Hydrex MV60 - 66
      ClHiTempRPMmA { S7_SetPoint := 'True'} : Real := 410.0;   // The max mA output in high temp reduced RPM mode
      CoolingFanTempC { S7_SetPoint := 'True'} : Real := 65.0;   // Temperature at which point cooling fan will turn on
      CoolingFanTimeOn { S7_SetPoint := 'True'} : Time := T#30S;   // The time the cooling fan will stay on for after temp below setpoint
      DrillTorqPotAlpha { S7_SetPoint := 'True'} : Real := 0.0;   // Low Pass Filter, Alpha be >= 0 and < 1. 0 No filterting.
      DrillThrottleAlpha { S7_SetPoint := 'True'} : Real := 0.0;   // Low Pass Filter, Alpha be >= 0 and < 1. 0 No filterting.
      DrillTorqLimLowPer { S7_SetPoint := 'True'} : Real := 80.0;   // Percent of Drill a torq Low Set point to allow before destroke flow for torq limit
      DrillTorqLimHighPer { S7_SetPoint := 'True'} : Real := 97.0;   // Percent of Drill a torq High Set point before destroke flow for torq limit
      DrillTorqLimTime { S7_SetPoint := 'True'} : Time := T#50MS;   // Debounce time that torq can be above low limit before limiting flow.
      DrillTorqLimSlewRise { S7_SetPoint := 'True'} : Real := 5.0;   // Rising Slew Rate mA/sec on Torq output not in Auto Mode
      DrillTorqLimSlewFall { S7_SetPoint := 'True'} : Real := 20.0;   // Falling Slew Rate mA/sec on Torq output not in Auto Mode
      FlushFlowFaultTime { S7_SetPoint := 'True'} : Time := T#10S;   // Time with flow while aux pump is running before fault
      HeartbeatTimeout { S7_SetPoint := 'True'} : Time := T#3S;   // Time heartbeat signal can remain unchanged before IO is dropped from remote console.
      HotOilFlowMinGPM { S7_SetPoint := 'True'} : Real := 5.0;   // Min Value of flow transducer
      HotOilFlowMaxGPM { S7_SetPoint := 'True'} : Real := 1000.0;   // MAx Value of flow transducer
      HotOilFlowAlpha { S7_SetPoint := 'True'} : Real := 0.0;   // Low Pass Filter, Alpha be >= 0 and < 1. 0 No filterting.
      HornOnTime { S7_SetPoint := 'True'} : Time := T#1S_500MS;   // Time horn output is on when horn requested
      HornSilenceTime { S7_SetPoint := 'True'} : Time := T#30S;   // Time horn will turn off if high temp shutdown
      HSLTShiftTime { S7_SetPoint := 'True'} : Time := T#2S;   // Time to allow system to shift before outputting to pump
      LampTestTime { S7_SetPoint := 'True'} : Time := T#2S;   // Time lamps will be on during lamp test
      LamptTestHornTime : Time := T#2S;   // Time horn will be on during lamp test
      LSHTShiftTime { S7_SetPoint := 'True'} : Time := T#4S;   // Time to allow system to shift before outputting to pump
      LubeFlowFaultTime { S7_SetPoint := 'True'} : Time := T#10S;   // Time After aux pump runnign before flow to be seen or alarm
      M1CurrentMin { S7_SetPoint := 'True'} : Real := 0.0;   // Min value of M1 Current Input- TBD actual values
      M1CurrentMax { S7_SetPoint := 'True'} : Real := 100.0;   // Max value of M1 Current Input- TBD actual values
      M1CurrentAlpha { S7_SetPoint := 'True'} : Real := 0.0;   // Low Pass Filter, Alpha be >= 0 and < 1. 0 No filterting.
      M2CurrentMin { S7_SetPoint := 'True'} : Real := 0.0;   // Min value of M2 Current Input- TBD actual values
      M2CurrentMax { S7_SetPoint := 'True'} : Real := 100.0;   // Max value of M2 Current Input - TBD actual values
      M2CurrentAlpha { S7_SetPoint := 'True'} : Real := 0.0;   // Low Pass Filter, Alpha be >= 0 and < 1. 0 No filterting.
      MotorFaultTime { S7_SetPoint := 'True'} : Time := T#15S;   // Time before signalling a motor fault if not started after start signal sent
      MUDoneTHper { S7_SetPoint := 'True'} : Real := 60.0;   // Torque threshold percent to determne mu done
      MUSpinAdjInc { S7_SetPoint := 'True'} : Real := 5.0;   // Increment in which the MU Spin value will adjust when requested
      MUSpinMaxSpeedPer { S7_SetPoint := 'True'} : Real := 80.0;   // The MU Spin max setting to limit user adjustment
      MUSpinTorqFtlbs { S7_SetPoint := 'True'} : Real := 2000.0;   // MU Spin torq settings. If Actual torq above this value spin complete
      MUTorqSlewRise { S7_SetPoint := 'True'} : Real := 45.0;   // Rising Slew Rate mA/sec on Torq output not in Auto Mode
      MUTorqSlewFall { S7_SetPoint := 'True'} : Real := 150.0;   // Falling Slew Rate mA/sec on Torq output not in Auto Mode
      MUFlowSlewRise { S7_SetPoint := 'True'} : Real := 25.0;   // Rising Slew Rate mA/sec on Flow Output
      MUFlowSlewFall { S7_SetPoint := 'True'} : Real := 150.0;   // Falling Slew Rate mA/sec on Flow Output
      MUFlowMinmA { S7_SetPoint := 'True'} : Real := 150.0;   // Min mA Output to Flow Pump in MU Torq
      MUFlowMaxmA { S7_SetPoint := 'True'} : Real := 800.0;   // Max mA Output to Flow Pump in MU Torq
      MUTorqPotAlpha { S7_SetPoint := 'True'} : Real := 0.0;   // Low Pass Filter, Alpha be >= 0 and < 1. 0 No filterting.
      OscMaxSpeedRPM { S7_SetPoint := 'True'} : Real := 30.0;   // Maximum rotary speed setpoint allowed for Oscialltor operation.
      OscMaxTorqFtLbs { S7_SetPoint := 'True'} : Real := 20000.0;   // Maximum torq setpoint allowed for Oscialltor operation.
      OscTorqLimLowPer { S7_SetPoint := 'True'} : Real := 90.0;   // Percent of Osc torq Low Set point to allow before destroke flow for torq limit
      OscTorqLimHighPer { S7_SetPoint := 'True'} : Real := 97.0;   // Percent of Osc torq High Set point before destroke flow for torq limit
      OscTorqLimTime { S7_SetPoint := 'True'} : Time := T#1MS;   // Debounce time that torq can be above low limit before limiting flow.
      PotZero { S7_SetPoint := 'True'} : Real := 5.0;   // Any percentage below this will be considered a zero input from the throttle.
      PumpOutMinmA { S7_SetPoint := 'True'} : Real := 200.0;   // Minimum mA setting to valve
      PumpOutMaxmA { S7_SetPoint := 'True'} : Real := 700.0;   // MaximummA setting to valve
      RotEncPPR { S7_SetPoint := 'True'} : Int := 22;   // Rotatry Encoder Counts per revolution
      RotStoppedTime { S7_SetPoint := 'True'} : Time := T#2S;   // Time without an encoder count before declaring stopped.
      SpeedLimLowRPM { S7_SetPoint := 'True'} : Real := 183.0;   // Speed limiter lower threshold
      SpeedLimHighRPM { S7_SetPoint := 'True'} : Real := 190.0;   // Speed limiter upper threshold
      SpeedLimSlewRise { S7_SetPoint := 'True'} : Real := 10.0;   // Rising Slew Rate mA/sec on Flow Output
      SpeedLimSlewFall { S7_SetPoint := 'True'} : Real := 10.0;   // Falling Slew Rate mA/sec on Flow Output
      SpinSpeedPer { S7_SetPoint := 'True'} : Real := 25.0;   // TheSpin speed setting in percent. User adjustable with Link Tilt. Value used for BO Spin also
      TDFwdPressMin { S7_SetPoint := 'True'} : Real := 0.0;   // Min value of TD Fwd Press transducer
      TDFwdPressMax { S7_SetPoint := 'True'} : Real := 5800.0;   // Max value of TD Fwd Press transducer
      TDFwdPressAlpha { S7_SetPoint := 'True'} : Real := 0.0;   // Low Pass Filter, Alpha be >= 0 and < 1. 0 No filterting.
      TDRevPressMax { S7_SetPoint := 'True'} : Real := 5800.0;   // Max value of TD Rev Press transducer
      TDRevPressMin { S7_SetPoint := 'True'} : Real := 0.0;   // Min value of TD Rev Press transducer
      TDRevPressAlpha { S7_SetPoint := 'True'} : Real := 0.0;   // Low Pass Filter, Alpha be >= 0 and < 1. 0 No filterting.
      TorqEFactorLow { S7_SetPoint := 'True'} : Real := 0.97;   // 0-1. Efficiency of Torque reading when below 5 RPM
      TorqEFactorHigh { S7_SetPoint := 'True'} : Real := 0.97;   // 0-1. Efficiency of Torque reading when below 5 RPM
      TorqInHSLT { S7_SetPoint := 'True'} : Real := 3.56;   // ft-lbs /psi in High speed low torque.
      TorqInLSHT { S7_SetPoint := 'True'} : Real := 7.119;   // ft-lbs / psi in low speed high torque.
      TorqPotMaxFtLbs { S7_SetPoint := 'True'} : Real := 30000.0;   // Max value in ft-lbs that the input pot should read(Actual value TBD)
      TorqOutExtraPSI { S7_SetPoint := 'True'} : Real := 51.60006;   // Extra PSI value added to torque output to overcome charge pressure
      TorqOutMinmA { S7_SetPoint := 'True'} : Real := 100.0;   // Minimum mA setting to valve
      TorqOutMaxmA { S7_SetPoint := 'True'} : Real := 800.0;   // MaximummA setting to valve
      TorqOutMinPSI { S7_SetPoint := 'True'} : Real := 0.0;   // Minimum PSI setting on Torq valve
      TorqOutMaxPSI { S7_SetPoint := 'True'} : Real := 5075.0;   // Maximum PSI setting on Torq Valve
      TorqOutHSLT { S7_SetPoint := 'True'} : Real := 3.56;   // ft-lbs /psi at output vavle in High speed low torque. Current values are same as Feedback actual value TBD
      TorqOutLSHT { S7_SetPoint := 'True'} : Real := 7.119;   // ft-lbs / psi output vavle in low speed high torque.Current values are same as Feedback actual value TBD
      TorqSetFactor { S7_SetPoint := 'True'} : Real := 1.0;   // Torq setpoint factor to increase the setpoint to ensure desired torq is reached. Torq limiting will be controlled via flow.
   END_VAR
BEGIN
END_DATA_BLOCK

ORGANIZATION_BLOCK "Main"   // OB1, LAD, ProgramCycle
TITLE = "Main Program Sweep (Cycle)"
{ S7_Optimized_Access := 'TRUE' }
// Bonanza Elect TD Rev0
// Written By Kristopher Gimenez January 16,2023
// For any questions please contact Automated Rig Technogies @ 403-723-6602
// This program is for the control the Bonanza Top drives utlizing the electric HPU.
// stored: SetENOAutomatically false
   VAR_INPUT
      Initial_Call : Bool;   // Initial call of this OB
      Remanence : Bool;   // =True, if remanent data are available
   END_VAR
   VAR_TEMP   // added for the SCL form of the ladder/FBD networks
      _w1 : Bool;
   END_VAR
BEGIN

REGION Network 2: Comm Checks, Communication is online after control system is powered up for 1min 10s. So to check when the system is full powered up
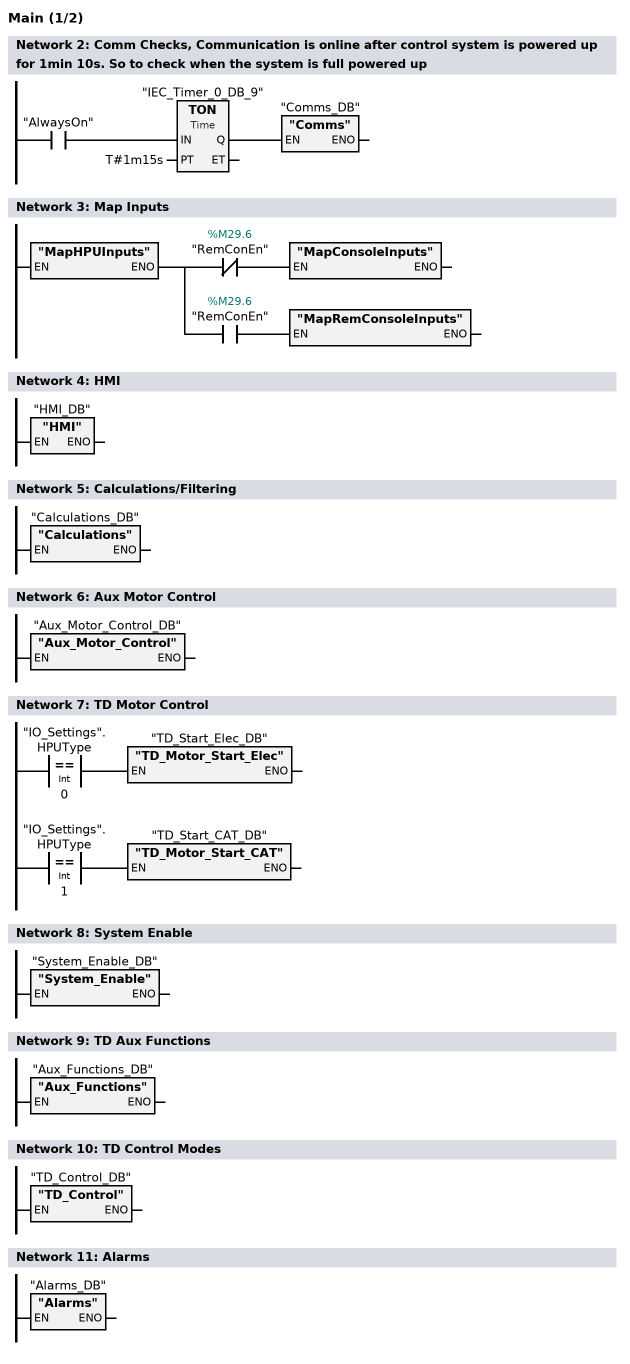
   RUNG wire#powerrail
      Contact( "AlwaysOn" )
      { S7_Templates := "time_type := Time" } "IEC_Timer_0_DB_9".TON(pt := T#1m15s, et =>)
      "Comms_DB"()
   END_RUNG
   // the same network as SCL:
   "IEC_Timer_0_DB_9".TON(IN := "AlwaysOn", PT := T#1m15s);
   IF "IEC_Timer_0_DB_9".Q THEN
       "Comms_DB"();   // "Comms"
   END_IF;
END_REGION

REGION Network 3: Map Inputs
   RUNG wire#powerrail
      "MapHPUInputs"()
      wire#w1
      I_Contact( "RemConEn" )
      "MapConsoleInputs"()
   END_RUNG
   RUNG wire#w1
      Contact( "RemConEn" )
      "MapRemConsoleInputs"()
   END_RUNG
   // the same network as SCL:
   "MapHPUInputs"(ENO => #_w1);
   IF #_w1 AND NOT "RemConEn" THEN "MapConsoleInputs"(); END_IF;
   IF #_w1 AND "RemConEn" THEN "MapRemConsoleInputs"(); END_IF;
END_REGION

REGION Network 4: HMI
   RUNG wire#powerrail
      "HMI_DB"()
   END_RUNG
   // the same network as SCL:
   "HMI_DB"();   // "HMI"
END_REGION

REGION Network 5: Calculations/Filtering
   RUNG wire#powerrail
      "Calculations_DB"()
   END_RUNG
   // the same network as SCL:
   "Calculations_DB"();   // "Calculations"
END_REGION

REGION Network 6: Aux Motor Control
   RUNG wire#powerrail
      "Aux_Motor_Control_DB"()
   END_RUNG
   // the same network as SCL:
   "Aux_Motor_Control_DB"();   // "Aux_Motor_Control"
END_REGION

REGION Network 7: TD Motor Control
   RUNG wire#powerrail
      { S7_Templates := "SrcType := Int" } EQ_Contact(in1 := "IO_Settings".HPUType, in2 := 0)
      "TD_Start_Elec_DB"()
   END_RUNG
   RUNG wire#powerrail
      { S7_Templates := "SrcType := Int" } EQ_Contact(in1 := "IO_Settings".HPUType, in2 := 1)
      "TD_Start_CAT_DB"()
   END_RUNG
   // the same network as SCL:
   IF "IO_Settings".HPUType = 0 THEN
       "TD_Start_Elec_DB"();   // "TD_Motor_Start_Elec"
   END_IF;
   IF "IO_Settings".HPUType = 1 THEN
       "TD_Start_CAT_DB"();   // "TD_Motor_Start_CAT"
   END_IF;
END_REGION

REGION Network 8: System Enable
   RUNG wire#powerrail
      "System_Enable_DB"()
   END_RUNG
   // the same network as SCL:
   "System_Enable_DB"();   // "System_Enable"
END_REGION

REGION Network 9: TD Aux Functions
   RUNG wire#powerrail
      "Aux_Functions_DB"()
   END_RUNG
   // the same network as SCL:
   "Aux_Functions_DB"();   // "Aux_Functions"
END_REGION

REGION Network 10: TD Control Modes
   RUNG wire#powerrail
      "TD_Control_DB"()
   END_RUNG
   // the same network as SCL:
   "TD_Control_DB"();   // "TD_Control"
END_REGION

REGION Network 11: Alarms
   RUNG wire#powerrail
      "Alarms_DB"()
   END_RUNG
   // the same network as SCL:
   "Alarms_DB"();   // "Alarms"
END_REGION

REGION Network 12: Indicators
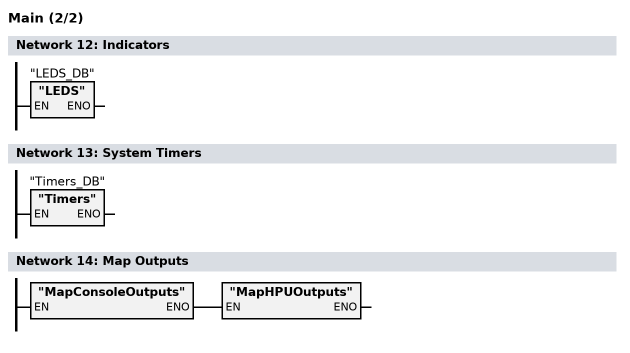
   RUNG wire#powerrail
      "LEDS_DB"()
   END_RUNG
   // the same network as SCL:
   "LEDS_DB"();   // "LEDS"
END_REGION

REGION Network 13: System Timers
   RUNG wire#powerrail
      "Timers_DB"()
   END_RUNG
   // the same network as SCL:
   "Timers_DB"();   // "Timers"
END_REGION

REGION Network 14: Map Outputs
   RUNG wire#powerrail
      "MapConsoleOutputs"()
      "MapHPUOutputs"()
   END_RUNG
   // the same network as SCL:
   "MapConsoleOutputs"(ENO => #_w1);
   IF #_w1 THEN "MapHPUOutputs"(); END_IF;
END_REGION
END_ORGANIZATION_BLOCK

FUNCTION_BLOCK "Comms"   // FB22, LAD
TITLE = COMMS
{ S7_Optimized_Access := 'TRUE' }
// Written By Kristopher Gimenez March 3rd ,2023
// 
// This block and its associated DB are used to poll the profinet network for device status.
// stored: AutoNumber false, MemoryReserve 100, SetENOAutomatically false
   VAR
      DeviceLADDR : HW_IOSYSTEM := 273;   // 273 from Hardware identifier of PN network
      DeviceMode : UInt;
      DeviceReturn : Int;
      DeviceStates : Array[0..1023] of Bool;
      DeviceFault : Array[0..1023] of Bool;
      HpuPlcStatus : Bool;
      HpuPlcOnline : Bool;
      ConRIOStatus : Bool;
      ConRIOOnline : Bool;
      HpuHmiStatus : Bool;
      HpuHmiOnline : Bool;
      ConHmiStatus : Bool;
      ConHmiOnline : Bool;
      DHHmiStatus : Bool;
      DHHmiOnline : Bool;
      CouplerStatus : Bool;
      CouplerOnline : Bool;
      RemHearbeatOK : Bool;
      HBOn_TON { S7_SetPoint := 'True'} : TON_TIME;
      HeatbeatLost { S7_SetPoint := 'True'} : Bool;
      HBOff_TON { S7_SetPoint := 'True'} : TON_TIME;
      HBPosTrig : Bool;
      HBNegTrig : Bool;
   END_VAR
   VAR_TEMP
      RetVal : Int;
      TimeZone : Time;
      HmiTemp : Bool;
      BusyStatus : Bool;
   END_VAR
   VAR_TEMP   // added for the SCL form of the ladder/FBD networks
      _w1 : Bool;
      _w2 : Bool;
   END_VAR
BEGIN

REGION Network 2: Read the PLC local Time, HMI get the time.
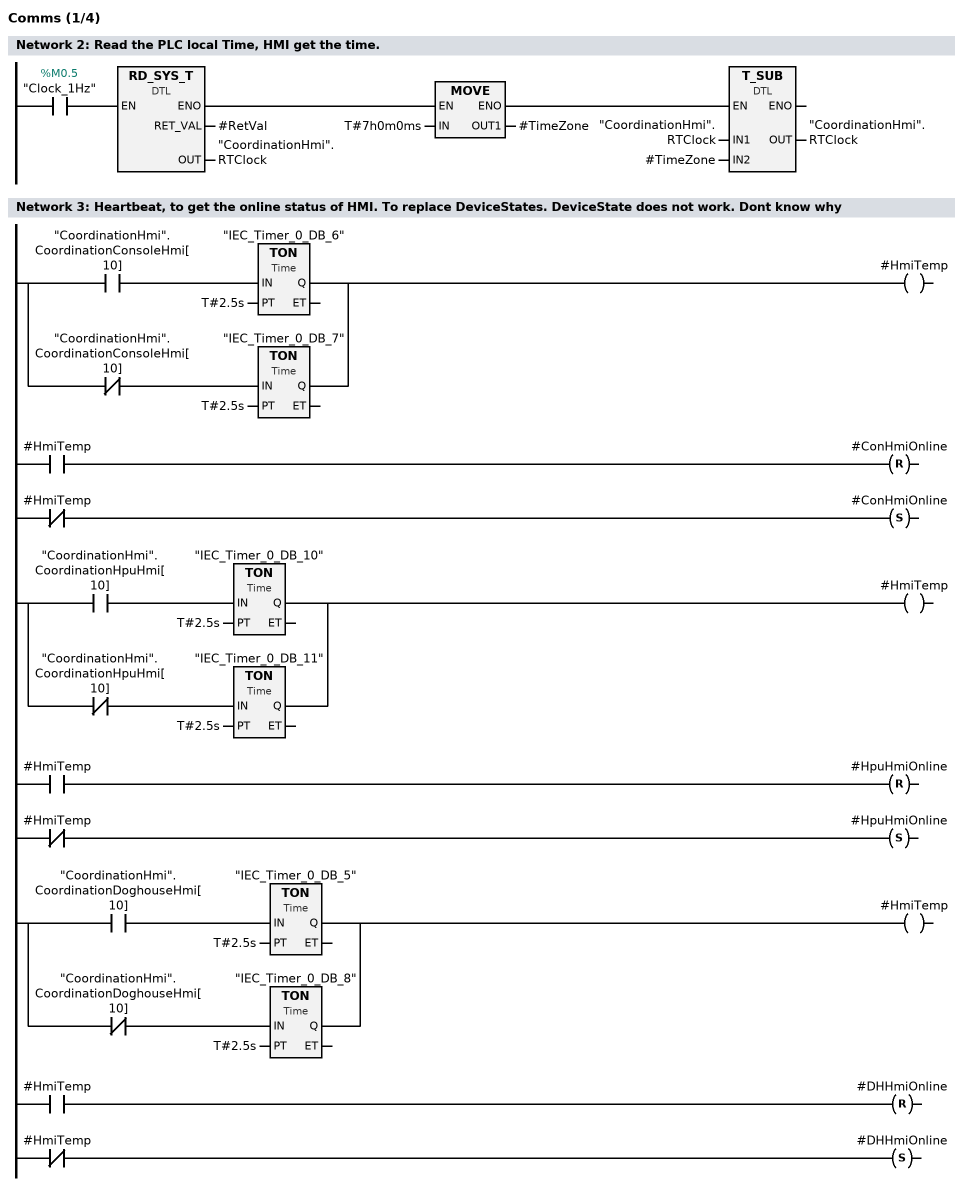
   RUNG wire#powerrail
      Contact( "Clock_1Hz" )
      { S7_Templates := "date_type := DTL" } RD_SYS_T(RET_VAL => #RetVal, OUT => "CoordinationHmi".RTClock)
      Move(in := T#7h0m0ms, out1 => #TimeZone)
      { S7_Templates := "[date_type := DTL, time_type := Time]" } T_SUB(IN1 := "CoordinationHmi".RTClock, IN2 := #TimeZone, OUT => "CoordinationHmi".RTClock)
   END_RUNG
   // the same network as SCL:
   #RetVal := RD_SYS_T(EN := "Clock_1Hz", OUT => "CoordinationHmi".RTClock, ENO => #_w1);
   IF #_w1 THEN
       #TimeZone := T#7h0m0ms;
       T_SUB(IN1 := "CoordinationHmi".RTClock, IN2 := #TimeZone, OUT => "CoordinationHmi".RTClock);
   END_IF;
END_REGION

REGION Network 3: Heartbeat, to get the online status of HMI. To replace DeviceStates. DeviceState does not work. Dont know why
   RUNG wire#powerrail
      Contact( "CoordinationHmi".CoordinationConsoleHmi[10] )
      { S7_Templates := "time_type := Time" } "IEC_Timer_0_DB_6".TON(pt := T#2.5s, et =>)
      wire#w1
      Coil( #HmiTemp )
   END_RUNG
   RUNG wire#powerrail
      I_Contact( "CoordinationHmi".CoordinationConsoleHmi[10] )
      { S7_Templates := "time_type := Time" } "IEC_Timer_0_DB_7".TON(pt := T#2.5s, et =>)
   END_RUNG wire#w1
   RUNG wire#powerrail
      Contact( #HmiTemp )
      R_Coil( #ConHmiOnline )
   END_RUNG
   RUNG wire#powerrail
      I_Contact( #HmiTemp )
      S_Coil( #ConHmiOnline )
   END_RUNG
   RUNG wire#powerrail
      Contact( "CoordinationHmi".CoordinationHpuHmi[10] )
      { S7_Templates := "time_type := Time" } "IEC_Timer_0_DB_10".TON(pt := T#2.5s, et =>)
      wire#w2
      Coil( #HmiTemp )
   END_RUNG
   RUNG wire#powerrail
      I_Contact( "CoordinationHmi".CoordinationHpuHmi[10] )
      { S7_Templates := "time_type := Time" } "IEC_Timer_0_DB_11".TON(pt := T#2.5s, et =>)
   END_RUNG wire#w2
   RUNG wire#powerrail
      Contact( #HmiTemp )
      R_Coil( #HpuHmiOnline )
   END_RUNG
   RUNG wire#powerrail
      I_Contact( #HmiTemp )
      S_Coil( #HpuHmiOnline )
   END_RUNG
   RUNG wire#powerrail
      Contact( "CoordinationHmi".CoordinationDoghouseHmi[10] )
      { S7_Templates := "time_type := Time" } "IEC_Timer_0_DB_5".TON(pt := T#2.5s, et =>)
      wire#w3
      Coil( #HmiTemp )
   END_RUNG
   RUNG wire#powerrail
      I_Contact( "CoordinationHmi".CoordinationDoghouseHmi[10] )
      { S7_Templates := "time_type := Time" } "IEC_Timer_0_DB_8".TON(pt := T#2.5s, et =>)
   END_RUNG wire#w3
   RUNG wire#powerrail
      Contact( #HmiTemp )
      R_Coil( #DHHmiOnline )
   END_RUNG
   RUNG wire#powerrail
      I_Contact( #HmiTemp )
      S_Coil( #DHHmiOnline )
   END_RUNG
   // the same network as SCL:
   "IEC_Timer_0_DB_6".TON(IN := "CoordinationHmi".CoordinationConsoleHmi[10], PT := T#2.5s);
   "IEC_Timer_0_DB_7".TON(IN := NOT "CoordinationHmi".CoordinationConsoleHmi[10], PT := T#2.5s);
   #HmiTemp := "IEC_Timer_0_DB_6".Q OR "IEC_Timer_0_DB_7".Q;
   IF #HmiTemp THEN #ConHmiOnline := FALSE; END_IF;
   IF NOT #HmiTemp THEN #ConHmiOnline := TRUE; END_IF;
   "IEC_Timer_0_DB_10".TON(IN := "CoordinationHmi".CoordinationHpuHmi[10], PT := T#2.5s);
   "IEC_Timer_0_DB_11".TON(IN := NOT "CoordinationHmi".CoordinationHpuHmi[10], PT := T#2.5s);
   #HmiTemp := "IEC_Timer_0_DB_10".Q OR "IEC_Timer_0_DB_11".Q;
   IF #HmiTemp THEN #HpuHmiOnline := FALSE; END_IF;
   IF NOT #HmiTemp THEN #HpuHmiOnline := TRUE; END_IF;
   "IEC_Timer_0_DB_5".TON(IN := "CoordinationHmi".CoordinationDoghouseHmi[10], PT := T#2.5s);
   "IEC_Timer_0_DB_8".TON(IN := NOT "CoordinationHmi".CoordinationDoghouseHmi[10], PT := T#2.5s);
   #HmiTemp := "IEC_Timer_0_DB_5".Q OR "IEC_Timer_0_DB_8".Q;
   IF #HmiTemp THEN #DHHmiOnline := FALSE; END_IF;
   IF NOT #HmiTemp THEN #DHHmiOnline := TRUE; END_IF;
END_REGION

REGION Network 4: Remote Console Heartbeat OK
   // Heartbeat is lost if state stays the same for the timeout time. Reset if Transition seen on heartbeat
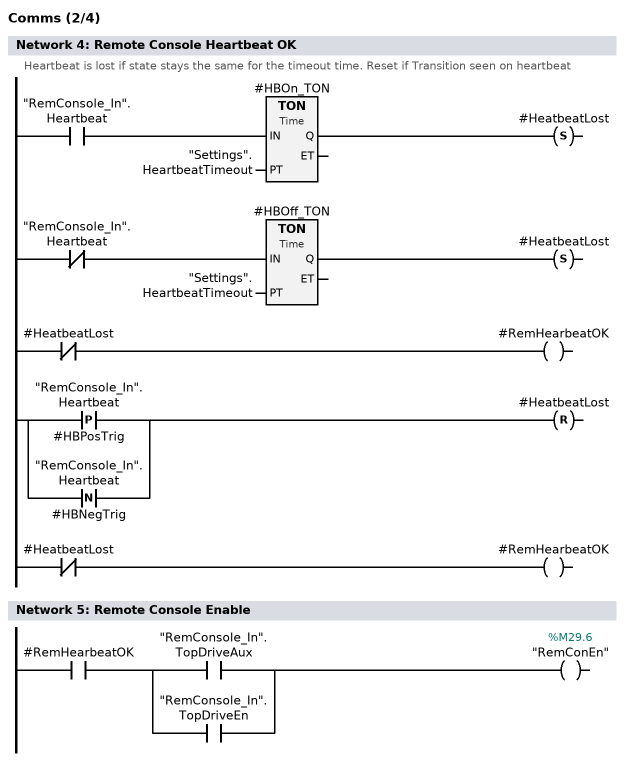
   RUNG wire#powerrail
      Contact( "RemConsole_In".Heartbeat )
      { S7_Templates := "time_type := Time" } #HBOn_TON.TON(pt := "Settings".HeartbeatTimeout, et =>)
      S_Coil( #HeatbeatLost )
   END_RUNG
   RUNG wire#powerrail
      I_Contact( "RemConsole_In".Heartbeat )
      { S7_Templates := "time_type := Time" } #HBOff_TON.TON(pt := "Settings".HeartbeatTimeout, et =>)
      S_Coil( #HeatbeatLost )
   END_RUNG
   RUNG wire#powerrail
      I_Contact( #HeatbeatLost )
      Coil( #RemHearbeatOK )
   END_RUNG
   RUNG wire#powerrail
      P_Contact(operand := "RemConsole_In".Heartbeat, bit := #HBPosTrig)
      wire#w1
      R_Coil( #HeatbeatLost )
   END_RUNG
   RUNG wire#powerrail
      N_Contact(operand := "RemConsole_In".Heartbeat, bit := #HBNegTrig)
   END_RUNG wire#w1
   RUNG wire#powerrail
      I_Contact( #HeatbeatLost )
      Coil( #RemHearbeatOK )
   END_RUNG
   // the same network as SCL:
   #HBOn_TON(IN := "RemConsole_In".Heartbeat, PT := "Settings".HeartbeatTimeout);   // TON
   IF #HBOn_TON.Q THEN #HeatbeatLost := TRUE; END_IF;
   #HBOff_TON(IN := NOT "RemConsole_In".Heartbeat, PT := "Settings".HeartbeatTimeout);   // TON
   IF #HBOff_TON.Q THEN #HeatbeatLost := TRUE; END_IF;
   #RemHearbeatOK := NOT #HeatbeatLost;
   #_w1 := "RemConsole_In".Heartbeat AND NOT #HBPosTrig;   // rising edge of "RemConsole_In".Heartbeat
   #HBPosTrig := "RemConsole_In".Heartbeat;
   #_w2 := NOT "RemConsole_In".Heartbeat AND #HBNegTrig;   // falling edge of "RemConsole_In".Heartbeat
   #HBNegTrig := "RemConsole_In".Heartbeat;
   IF #_w1 OR #_w2 THEN #HeatbeatLost := FALSE; END_IF;
   #RemHearbeatOK := NOT #HeatbeatLost;
END_REGION

REGION Network 5: Remote Console Enable
   RUNG wire#powerrail
      Contact( #RemHearbeatOK )
      wire#w1
      Contact( "RemConsole_In".TopDriveAux )
      wire#w2
      Coil( "RemConEn" )
   END_RUNG
   RUNG wire#w1
      Contact( "RemConsole_In".TopDriveEn )
   END_RUNG wire#w2
   // the same network as SCL:
   "RemConEn" := #RemHearbeatOK AND ("RemConsole_In".TopDriveAux OR "RemConsole_In".TopDriveEn);
END_REGION

REGION Network 6: Comms
   // Perform Device Exist check (mode 4) to see if device online
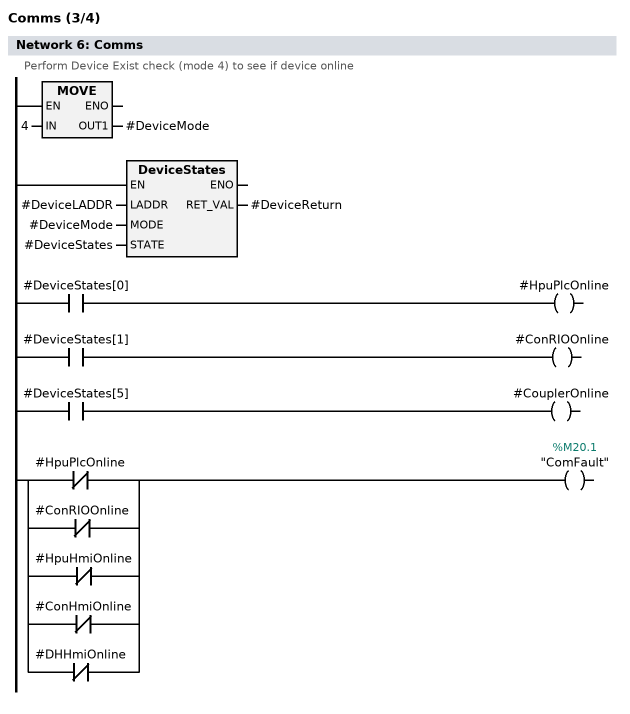
   RUNG wire#powerrail
      Move(in := 4, out1 => #DeviceMode)
   END_RUNG
   RUNG wire#powerrail
      DeviceStates(LADDR := #DeviceLADDR, MODE := #DeviceMode, STATE := #DeviceStates, Ret_Val => #DeviceReturn)
   END_RUNG
   RUNG wire#powerrail
      Contact( #DeviceStates[0] )
      Coil( #HpuPlcOnline )
   END_RUNG
   RUNG wire#powerrail
      Contact( #DeviceStates[1] )
      Coil( #ConRIOOnline )
   END_RUNG
   RUNG wire#powerrail
      Contact( #DeviceStates[5] )
      Coil( #CouplerOnline )
   END_RUNG
   RUNG wire#powerrail
      I_Contact( #HpuPlcOnline )
      wire#w1
      Coil( "ComFault" )
   END_RUNG
   RUNG wire#powerrail
      I_Contact( #ConRIOOnline )
   END_RUNG wire#w1
   RUNG wire#powerrail
      I_Contact( #HpuHmiOnline )
   END_RUNG wire#w1
   RUNG wire#powerrail
      I_Contact( #ConHmiOnline )
   END_RUNG wire#w1
   RUNG wire#powerrail
      I_Contact( #DHHmiOnline )
   END_RUNG wire#w1
   // the same network as SCL:
   #DeviceMode := 4;
   #DeviceReturn := DeviceStates(LADDR := #DeviceLADDR, MODE := #DeviceMode, STATE := #DeviceStates);
   #HpuPlcOnline := #DeviceStates[0];
   #ConRIOOnline := #DeviceStates[1];
   #CouplerOnline := #DeviceStates[5];
   "ComFault" := NOT #HpuPlcOnline OR NOT #ConRIOOnline OR NOT #HpuHmiOnline OR NOT #ConHmiOnline OR NOT #DHHmiOnline;
END_REGION

REGION Network 7: Fault State
   // Perform Device Fault check (mode 2) to see if device has fault. Set Status as Opposite. 1 = No Fault
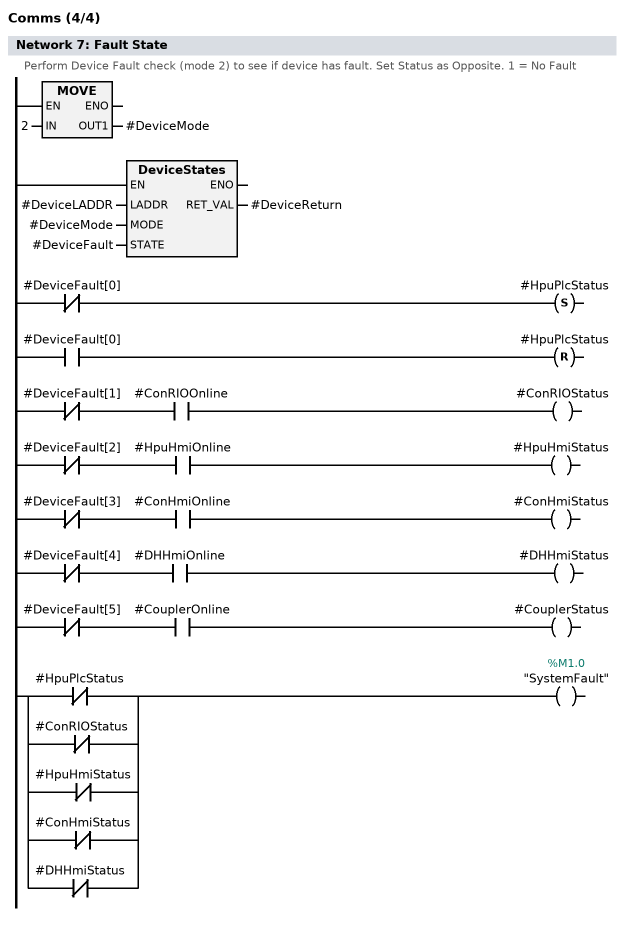
   RUNG wire#powerrail
      Move(in := 2, out1 => #DeviceMode)
   END_RUNG
   RUNG wire#powerrail
      DeviceStates(LADDR := #DeviceLADDR, MODE := #DeviceMode, STATE := #DeviceFault, Ret_Val => #DeviceReturn)
   END_RUNG
   RUNG wire#powerrail
      I_Contact( #DeviceFault[0] )
      S_Coil( #HpuPlcStatus )
   END_RUNG
   RUNG wire#powerrail
      Contact( #DeviceFault[0] )
      R_Coil( #HpuPlcStatus )
   END_RUNG
   RUNG wire#powerrail
      I_Contact( #DeviceFault[1] )
      Contact( #ConRIOOnline )
      Coil( #ConRIOStatus )
   END_RUNG
   RUNG wire#powerrail
      I_Contact( #DeviceFault[2] )
      Contact( #HpuHmiOnline )
      Coil( #HpuHmiStatus )
   END_RUNG
   RUNG wire#powerrail
      I_Contact( #DeviceFault[3] )
      Contact( #ConHmiOnline )
      Coil( #ConHmiStatus )
   END_RUNG
   RUNG wire#powerrail
      I_Contact( #DeviceFault[4] )
      Contact( #DHHmiOnline )
      Coil( #DHHmiStatus )
   END_RUNG
   RUNG wire#powerrail
      I_Contact( #DeviceFault[5] )
      Contact( #CouplerOnline )
      Coil( #CouplerStatus )
   END_RUNG
   RUNG wire#powerrail
      I_Contact( #HpuPlcStatus )
      wire#w1
      Coil( "SystemFault" )
   END_RUNG
   RUNG wire#powerrail
      I_Contact( #ConRIOStatus )
   END_RUNG wire#w1
   RUNG wire#powerrail
      I_Contact( #HpuHmiStatus )
   END_RUNG wire#w1
   RUNG wire#powerrail
      I_Contact( #ConHmiStatus )
   END_RUNG wire#w1
   RUNG wire#powerrail
      I_Contact( #DHHmiStatus )
   END_RUNG wire#w1
   // the same network as SCL:
   #DeviceMode := 2;
   #DeviceReturn := DeviceStates(LADDR := #DeviceLADDR, MODE := #DeviceMode, STATE := #DeviceFault);
   IF NOT #DeviceFault[0] THEN #HpuPlcStatus := TRUE; END_IF;
   IF #DeviceFault[0] THEN #HpuPlcStatus := FALSE; END_IF;
   #ConRIOStatus := NOT #DeviceFault[1] AND #ConRIOOnline;
   #HpuHmiStatus := NOT #DeviceFault[2] AND #HpuHmiOnline;
   #ConHmiStatus := NOT #DeviceFault[3] AND #ConHmiOnline;
   #DHHmiStatus := NOT #DeviceFault[4] AND #DHHmiOnline;
   #CouplerStatus := NOT #DeviceFault[5] AND #CouplerOnline;
   "SystemFault" := NOT #HpuPlcStatus OR NOT #ConRIOStatus OR NOT #HpuHmiStatus OR NOT #ConHmiStatus OR NOT #DHHmiStatus;
END_REGION
END_FUNCTION_BLOCK

FUNCTION "MapHPUInputs" : Void
{ S7_Optimized_Access := 'TRUE' }
VERSION : 0.1
   VAR_TEMP 
      TempSpeed1 : Real;
      LastCount : DInt;
      tempgate : Bool;
      Tempready : Bool;
      Tempmask : DInt;
      TempMeasured : Real;
      Tempulint : ULInt;
      Temp77 : Bool;
      Tempzzero : Bool;
      CalcSpeed : DInt;
   END_VAR


BEGIN
	(* #MapHPUInputs Written BY Kristopher Gimenez January 19,2023
	This block is will map the input variables and convert raw signals into measured values
	*)
	
	//HPU Slot2 TM Count Encoder Input
	"RotaryCounts" := "HPU_In".Slot2.COUNT_VALUE;
	//#CalcSpeed := 60*("RotaryCounts" - "LastCount") / 22;
	//"LastCount" :="RotaryCounts";
	
	//"RotaryRPM" := "HPU_In".Slot2.MEASURED_VALUE;
	//#Tempulint := 1;
	//IF "HPU_In".Slot2.MEASURED_VALUE > 0 THEN
	//    #TempMeasured := ("HPU_In".Slot2.MEASURED_VALUE - 1000000000.0) / 1000000.0;
	//ELSE
	//    #TempMeasured := 0;
	//END_IF;
	//IF "HPU_In".Slot2.MEASURED_VALUE > 0 THEN
	//    #TempSpeed1 := (#TempMeasured - 85) * 5.7037037037;
	//ELSE
	//    #TempSpeed1 := 0;
	//END_IF;
	"RotEncOvFl" := "HPU_In".Slot2.EVENT_OFLW;
	"RotEncUnFl" := "HPU_In".Slot2.EVENT_UFLW;
	"RotEncA" := "HPU_In".Slot2.STS_DI0;
	"RotEncB" := "HPU_In".Slot2.STS_DI1;
	#tempgate := "HPU_In".Slot2.STS_SW_GATE;
	#Tempready := "HPU_In".Slot2.STS_READY;
	#Tempzzero := "HPU_In".Slot2.EVENT_ZERO;
	#Temp77 := "HPU_In".Slot2.LD_ERROR;
	//HPU Slot 3 - 16 x DI
	"AuxPumpRunning" := "HPU_In".Slot3.Ch0;
	"CoolingFanRunning"  :="HPU_In".Slot3.Ch1;
	"M1Running" := "HPU_In".Slot3.Ch2;
	"M2Running" := "HPU_In".Slot3.Ch3;
	"AuxPumpHOA":= "HPU_In".Slot3.Ch4;
	"CoolingFanHOA" := "HPU_In".Slot3.Ch5;
	"M1HOA" := "HPU_In".Slot3.Ch6;
	"M2HOA" :="HPU_In".Slot3.Ch7;
	"TDFlushFlowSw":= "HPU_In".Slot3.Ch8;
	"TDLubeFlowSw":= "HPU_In".Slot3.Ch9;
	"ChargePump1PSw" := "HPU_In".Slot3.Ch10;
	"ChargePump2PSw" := "HPU_In".Slot3.Ch11;
	
	//HPU Slot 4 - 16 x DI
	"TankLowLevelSw" := "HPU_In".Slot4.Ch0;
	"TankHighTempSw" :="HPU_In".Slot4.Ch1;
	"TDFwdFilter1" := "HPU_In".Slot4.Ch2;
	"TDFwdFilter2" := "HPU_In".Slot4.Ch3;
	"TDRevFilter1":= "HPU_In".Slot4.Ch4;
	"TDRevFilter2" := "HPU_In".Slot4.Ch5;
	"AuxReturnFilter" := "HPU_In".Slot4.Ch6;
	"KLoopFilter" := "HPU_In".Slot4.Ch7;
	"ChargeFilter" := 0;//"HPU_In".Slot4.Ch8;
	"ElevClFeedback" := 0;// "HPU_In".Slot4.Ch9;
	 
	 //HPU Slot 5 8 x AI U
	"M1CurrentRaw" := "HPU_In".Slot5.Ch0;
	"M1CurrentV" := "AiV_Raw2V"("M1CurrentRaw");
	"M2CurrentRaw" := "HPU_In".Slot5.Ch1;
	"M2CurrentV" := "AiV_Raw2V"("M2CurrentRaw");
	"HPU_AiV2SpareRaw" :="HPU_In".Slot5.Ch2;
	"HPU_AiV2SpareV"  := "AiV_Raw2V"("HPU_AiV2SpareRaw" );
	"HPU_AiV3SpareRaw" := "HPU_In".Slot5.Ch3;
	"HPU_AiV3SpareV" := "AiV_Raw2V"("HPU_AiV3SpareRaw");
	"HPU_AiV4SpareRaw" := "HPU_In".Slot5.Ch4;
	"HPU_AiV4SpareV" := "AiV_Raw2V"("HPU_AiV4SpareRaw");
	"HPU_AiV5SpareRaw" := "HPU_In".Slot5.Ch5;
	"HPU_AiV5SpareV" := "AiV_Raw2V"("HPU_AiV5SpareRaw");
	"HPU_AiV6SpareRaw" := "HPU_In".Slot5.Ch6;
	"HPU_AiV6SpareV" := "AiV_Raw2V"("HPU_AiV6SpareRaw");
	"HPU_AiV7SpareRaw" := "HPU_In".Slot5.Ch7;
	"HPU_AiV7SpareV" := "AiV_Raw2V"("HPU_AiV7SpareRaw");
	
	
	//HPU Slot 6 8 x AI 4-20ma
	"TDPressFWDRaw" := "HPU_In".Slot6.Ch0;
	"TDPressFWDmA" := "AiV_Raw2mA"("TDPressFWDRaw");
	"TDPressREVRaw" := "HPU_In".Slot6.Ch1;
	"TDPressREVmA" := "AiV_Raw2mA"("TDPressREVRaw");
	"ClosedLoopTempRaw" := "HPU_In".Slot6.Ch2;
	"ClosedLoopTempmA" := "AiV_Raw2mA"("ClosedLoopTempRaw");
	"ChargeFlowRaw" := "HPU_In".Slot6.Ch3;
	"ChargeFlowmA" := "AiV_Raw2mA"("ChargeFlowRaw");
	"HotOilShuttleFlowRaw" := "HPU_In".Slot6.Ch4;
	"HotOilShuttleFlowmA" := "AiV_Raw2mA"("HotOilShuttleFlowRaw");
	"AuxFlowRaw" := "HPU_In".Slot6.Ch5;
	"AuxFlowmA" := "AiV_Raw2mA"("AuxFlowRaw");
	"ChargePress1Raw" := "HPU_In".Slot6.Ch6;
	"ChargePress1mA" := "AiV_Raw2mA"("ChargePress1Raw");
	"ChargePress2Raw" := "HPU_In".Slot6.Ch7;
	"ChargePress2mA" := "AiV_Raw2mA"("ChargePress2Raw");
	
	
	//Slot 7 TM Pulse status inputs
	"TDP1FwdCmdActRaw" := "HPU_In".Slot7.Ch0.MEASURE_CURRENT;
	"TDP1FwdCmdActmA" := "TM_Pulse_Raw2mA"("TDP1FwdCmdActRaw");
	"TDP1RevCmdActRaw" := "HPU_In".Slot7.Ch1.MEASURE_CURRENT;
	"TDP1RevCmdActmA" := "TM_Pulse_Raw2mA"("TDP1RevCmdActRaw");
	
	
	//Slot 8 TM Pulse status inputs
	"TDP2FwdCmdActRaw" := "HPU_In".Slot8.Ch0.MEASURE_CURRENT;
	"TDP2FwdCmdActmA" := "TM_Pulse_Raw2mA"("TDP2FwdCmdActRaw");
	"TDP2RevCmdActRaw" := "HPU_In".Slot8.Ch1.MEASURE_CURRENT;
	"TDP2RevCmdActmA" := "TM_Pulse_Raw2mA"("TDP2RevCmdActRaw");
	
	//Slot 9 TM Pulse status inputs
	"TDTorqCmdActRaw" :="HPU_In".Slot9.Ch0.MEASURE_CURRENT;
	"TDTorqCmdActmA":="TM_Pulse_Raw2mA"("TDTorqCmdActRaw");
	
	
	
	
END_FUNCTION

FUNCTION "AiV_Raw2V" : Real
{ S7_Optimized_Access := 'TRUE' }
VERSION : 0.1
   VAR_INPUT 
      RawInput : Int;
   END_VAR


BEGIN
	(* #AiV_Raw2V Written BY Kristopher Gimenez January 19,2023
	This block is used to convert the Raw voltage input signal to a V for Unipolar 0-10 V inputs setup. Note 10V = 27648. 
	*)
	
	
	#AiV_Raw2V := INT_TO_REAL(#RawInput) / 27648.0 * 10;
	
	
END_FUNCTION

FUNCTION "AiV_Raw2mA" : Real
{ S7_Optimized_Access := 'TRUE' }
VERSION : 0.1
   VAR_INPUT 
      RawInput : Int;
   END_VAR


BEGIN
	(* #AiV_Raw2mA Written BY Kristopher Gimenez January 19,2023
	This block is used to convert the Raw mA input signal to a mA for Unipolar 4-20ma inputs setup. 
	Note 100% signal = 20mA = 27648. 
	*)
	
	
	#AiV_Raw2mA := (INT_TO_REAL(#RawInput) / 27648.0 * 16.0)+4.0;
	
	
END_FUNCTION

FUNCTION "TM_Pulse_Raw2mA" : Real
{ S7_Optimized_Access := 'TRUE' }
VERSION : 0.1
   VAR_INPUT 
      RawInput : Int;
   END_VAR


BEGIN
	(* TM_Pulse_Raw2mA Written BY Kristopher Gimenez January 19,2023
	This block is used to convert the Raw current input(measured output) to a ma for 2CH TM pulse module. Note 2A = 27648. 
	*)
	
	
	#TM_Pulse_Raw2mA := INT_TO_REAL(#RawInput) / 27648.0 * 2000;
	
END_FUNCTION

FUNCTION "MapConsoleInputs" : Void
{ S7_Optimized_Access := 'TRUE' }
VERSION : 0.1

BEGIN
	(* #MapHPUConsoleInputs Written BY Kristopher Gimenez January 19,2023
	This block is will map the input variables for the console dependant on whether a third part connection is made. It will also convert raw signals into measured values for the console inputs. 
	*)
	
	(*
	//To be Added Here
	If Remote Console connect heartbeat OK, Remote Enable is On and Local Console Off use remote console values. 
	*)
	
	//Slot 1 16 x DI
	"LinkRetSw" := "Console_In".Slot1.Ch0;
	"TDAuxSw":= "Console_In".Slot1.Ch1;
	"LinkExtSw":= "Console_In".Slot1.Ch2;
	"TDEnSW":= "Console_In".Slot1.Ch3;
	"HSLT_Sw":= "Console_In".Slot1.Ch4;
	"HandlerFwdSw":= "Console_In".Slot1.Ch5;
	"HandlerRevSw":= "Console_In".Slot1.Ch6;
	"MPNotRunning" := NOT "Console_In".Slot1.Ch7;//
	"QuillLockSw":= "Console_In".Slot1.Ch8;
	"BUWClSw":= "Console_In".Slot1.Ch9;
	"BUWDnSw":= "Console_In".Slot1.Ch10;
	"BUWUpSw":= "Console_In".Slot1.Ch11;
	"TDModeMUSpinSw":= "Console_In".Slot1.Ch12;
	"TDModeMUTorqSw":= "Console_In".Slot1.Ch13;
	"TDModeDrillRevSw":= "Console_In".Slot1.Ch14;
	"TDModeBreakOutSw":= "Console_In".Slot1.Ch15;
	
	//Slot 2 16 x DI
	"ElevOpSw" := "Console_In".Slot2.Ch0;
	"TDExtSw" := "Console_In".Slot2.Ch1;
	"ElevClSw" := "Console_In".Slot2.Ch2;
	"TDRetSw":= "Console_In".Slot2.Ch3;
	"PTO_Sw" := "Console_In".Slot2.Ch4;
	"PurgePressureSw":= "Console_In".Slot2.Ch5;
	"MSVClSw":= "Console_In".Slot2.Ch6;
	"MSVAutoSw" := "Console_In".Slot2.Ch7;
	"MSVOpSw" := "Console_In".Slot2.Ch8;
	"LinkFloatSw":= "Console_In".Slot2.Ch9;
	
	//Slot 3 AI 8 xU
	"MUTorqPotRaw" := "Console_In".Slot3.Ch0;
	"MUTorqPotV" := "AiV_Raw2V"("MUTorqPotRaw");
	"DrillTorqPotRaw" := "Console_In".Slot3.Ch1;
	"DrillTorqPotV" := "AiV_Raw2V"("DrillTorqPotRaw");
	"DrillThrottlePotRaw" := "Console_In".Slot3.Ch2;
	"DrillThrottlePotV" := "AiV_Raw2V"("DrillThrottlePotRaw");
	"Con_AiV3SpareRaw" :=  "Console_In".Slot3.Ch3;
	"Con_AiV3SpareV" := "AiV_Raw2V"("Con_AiV3SpareRaw");
	"Con_AiV4SpareRaw" :=  "Console_In".Slot3.Ch4;
	"Con_AiV4SpareV" := "AiV_Raw2V"("Con_AiV4SpareRaw");
	"Con_AiV5SpareRaw" :=  "Console_In".Slot3.Ch5;
	"Con_AiV5SpareV" := "AiV_Raw2V"("Con_AiV5SpareRaw");
	"Con_AiV6SpareRaw" :=  "Console_In".Slot3.Ch6;
	"Con_AiV6SpareV" := "AiV_Raw2V"("Con_AiV6SpareRaw");
	"Con_AiV7SpareRaw" :=  "Console_In".Slot3.Ch7;
	"Con_AiV7SpareV" := "AiV_Raw2V"("Con_AiV7SpareRaw");
	
	
	
	
	
END_FUNCTION

FUNCTION "MapRemConsoleInputs" : Void
{ S7_Optimized_Access := 'TRUE' }
VERSION : 0.1

BEGIN
	(* #MapHPUConsoleInputs Written BY Kristopher Gimenez January 19,2023
	This block is will map the input variables for the console dependant on whether a third part connection is made. It will also convert raw signals into measured values for the console inputs. 
	*)
	
	(*
	//To be Added Here
	If Remote Console connect heartbeat OK, Remote Enable is On and Local Console Off use remote console values. 
	*)
	
	//Digital Inputs
	"LinkRetSw" := "RemConsole_In".LinkTiltRetr;
	"TDAuxSw":= "RemConsole_In".TopDriveAux;
	"LinkExtSw":= "RemConsole_In".LinkTiltExt;
	"TDEnSW":= "RemConsole_In".TopDriveEn;
	"HSLT_Sw":= "RemConsole_In".HSLTEn;
	"HandlerFwdSw":= "RemConsole_In".HandlerFwd;
	"HandlerRevSw":= "RemConsole_In".HandlerRev;
	"MPNotRunning":= "RemConsole_In".MudPumpRunning;
	"QuillLockSw":= "RemConsole_In".QuillLock;
	"BUWClSw":= "RemConsole_In".BUWClose;
	"BUWDnSw":= "RemConsole_In".BUWDown;
	"BUWUpSw":= "RemConsole_In".BUWUp;
	"TDModeMUSpinSw":= "RemConsole_In".TDModeMUSpin;
	"TDModeMUTorqSw":= "RemConsole_In".TDModeMUTorq;
	"TDModeDrillRevSw":= "RemConsole_In".TDModeRev;
	"TDModeBreakOutSw":= "RemConsole_In".TDModeBO;
	"ElevOpSw" := "RemConsole_In".ElevOp;
	"TDExtSw":= "RemConsole_In".TDExt;
	"ElevClSw":= "RemConsole_In".ElevCl;
	"TDRetSw":= "RemConsole_In".TDRet;
	"PTO_Sw":= "RemConsole_In".PTO;
	"MSVClSw":= "RemConsole_In".MSVClose;
	"MSVAutoSw":= "RemConsole_In".MSVAuto;
	"MSVOpSw":= "RemConsole_In".MSVOpen;
	"LinkFloatSw":= "RemConsole_In".LinkTiltFloat;
	
	//Analog Inputs
	"MUTorqPotRaw" := "RemConsole_In".MUTorqLim;
	"MUTorqPotV" := "AiV_Raw2V"("MUTorqPotRaw");
	"DrillTorqPotRaw" := "RemConsole_In".DrillTorqLim;
	"DrillTorqPotV" := "AiV_Raw2V"("DrillThrottlePotRaw");
	"DrillThrottlePotRaw" := "RemConsole_In".DrillThrottle;
	"DrillThrottlePotV" := "AiV_Raw2V"("DrillThrottlePotRaw");
	
	
	
	
	
	
END_FUNCTION

FUNCTION_BLOCK "HMI"   // FB20, LAD
TITLE = HMI
{ S7_Optimized_Access := 'TRUE' }
// Bonanza Elect TD Rev0
// Written By Kristopher Gimenez Feb 13,2023
// 
// This block and its associated DB are used for HMI specific actions, interlocks and visualizations.
// stored: AutoNumber false, MemoryReserve 100, SetENOAutomatically false
   VAR
      DHScreen : Array[0..4] of Int;   // Current Info of the Doghouse HMI
      HPUScreen : Array[0..4] of Int;   // Current Info Number of the HPU HMI
      ConsoleScreen : Array[0..4] of Int;   // Current Info Number of the Console HMI
      OscEnable : Bool;   // Oscillator Enable Bit. Set on HMI
      OscAllowEn : Bool;   // Allow Enable from HMI screen.
   END_VAR
   VAR RETAIN
      OscBumpAdj { S7_SetPoint := 'True'} : Real := 20.0;   // Amount the bump position will adjust if increment/decremented. Set on HMI
   END_VAR
   VAR
      OscBumpFwdInc : Bool;   // Used to increase the Fwd Bump by the adjust amount
      OscBumpFwdDec : Bool;   // Used to dec the Fwd Bump by the adjust amount
      OscBumpReactive : Bool;   // Used to trigger Reactive Bump. Always FWD
      OscBumpRevInc : Bool;   // Used to increase the RevBump by the adjust amount
      OscBumpRevDec : Bool;   // Used to dec the Rev Bump by the adjust amount
      OscBumpFwd : Bool;   // Bit used to increase the Home position
      OscBumpRev : Bool;   // Bit used to decrease the home position
   END_VAR
   VAR RETAIN
      OscBumpFwdDeg : Real;   // Amount of Degrees to Bump Forward
      OscBumpRevDeg : Real;   // Amount of Degress to Bump in Rev
   END_VAR
   VAR
      OscHoldButton : Bool;   // Bit used to change color of Button On HMI
      OscHold : Bool;   // Bit used to hold Osc at current position.
      OscBumpFwdButton : Bool;
      OscBumpRevButton : Bool;
      OscBumpFwdRevButtonEn : Bool;
      OscHomeRelDeg : Real;   // Relative Oscillator Home position in degrees.
   END_VAR
   VAR RETAIN
      OscP1FwdMinmA { S7_SetPoint := 'True'} : Real := 200.0;   // Min mA output for Osc FWD on P1
      OscP1FwdMaxmA { S7_SetPoint := 'True'} : Real := 600.0;   // Max mA output for Osc FWD on P1
      OscP1RevMinmA { S7_SetPoint := 'True'} : Real := 200.0;   // Min mA output for Osc Rev on P1
      OscP1RevMaxmA { S7_SetPoint := 'True'} : Real := 600.0;   // Max mA output for Osc Rev on P1
      OscP1HoldmA { S7_SetPoint := 'True'} : Real := 300.0;   // mA Setting to hold position while oscillating
      OscP2FwdMinmA { S7_SetPoint := 'True'} : Real := 200.0;   // Min mA output for Osc FWD on P2
      OscP2FwdMaxmA { S7_SetPoint := 'True'} : Real := 600.0;   // Max mA output for Osc FWD on P2
      OscP2RevMinmA { S7_SetPoint := 'True'} : Real := 200.0;   // Min mA output for Osc Rev on P2
      OscP2RevMaxmA { S7_SetPoint := 'True'} : Real := 600.0;   // Max mA output for Osc Rev on P2
      OscP2HoldmA { S7_SetPoint := 'True'} : Real := 300.0;   // mA Setting to hold position while oscillating
   END_VAR
   VAR
      OscPosZero : Bool;   // Bit used toset the current rotary position as zero degrees and reset Home.
   END_VAR
   VAR RETAIN
      OscSlewRiseFast { S7_SetPoint := 'True'} : Real := 100.0;   // Rising Slew Rate mA/sec for Flow, fast reaction
      OscSlewRiseSlow { S7_SetPoint := 'True'} : Real := 10.0;   // Rising Slew Rate mA/sec on Flow, slow reaction
      OscSlewFallFast { S7_SetPoint := 'True'} : Real := 100.0;   // Falling Slew Rate mA/sec for Flow, fast reaction
      OscSlewFallSlow { S7_SetPoint := 'True'} : Real := 10.0;   // Falling Slew Rate mA/sec on Flow, slow reaction
      OscSpeedTHper { S7_SetPoint := 'True'} : Real := 75.0;   // Speed threshold percent to determine fast or slow slew rates
      OscSpeedHoldper { S7_SetPoint := 'True'} : Real := 95.0;   // Speed threshold percent to where control is held.
      OscSpeedFwdRPM { S7_SetPoint := 'True'} : Real := 15.0;   // Osc FWD speed setpoint. Set on HMI
      OscSpeedRevRPM { S7_SetPoint := 'True'} : Real := 15.0;   // Osc Rev speed setpoint Set on HMI
   END_VAR
   VAR
      OscSpeedFwdZone1 : Real;   // Calc value base on Input and TH percent. Below this speed setpoint - fast ramp up to the speed
      OscSpeedFwdZone2 : Real;   // Calc value base on Input and TH percent, Between Set 1 and Set 2 - Slow ramp up to speed
      OscSpeedFwdZone3 : Real;   // Calc value base on Input and TH percent,Between Set 2 and Set 3 - Maintina Speed
      OscSpeedFwdZone4 : Real;   // Calc value base on Input and TH percent,Between Set 3 and 4 - Slow Ramp Down. Above this speed Fast ramp down
      OscSpeedRevZone1 : Real;   // Calc value base on Input and TH percent. Below this speed setpoint - fast ramp up to the speed
      OscSpeedRevZone2 : Real;   // Calc value base on Input and TH percent, Between Set 1 and Set 2 - Slow ramp up to speed
      OscSpeedRevZone3 : Real;   // Calc value base on Input and TH percent,Between Set 2 and Set 3 - Maintina Speed
      OscSpeedRevZone4 : Real;   // Calc value base on Input and TH percent,Between Set 3 and 4 - Slow Ramp Down. Above this speed Fast ramp down
      OscStart : Bool;   // Bit used to start Oscillating
      OscStartButton : Bool;   // Bit used to change color of Button On HMI
      OscStop : Bool;   // Bit used to Stop Oscillating or Holding
      OscStopButton : Bool;   // Bit used to change color of Button On HMI
   END_VAR
   VAR RETAIN
      OscTorqAdj { S7_SetPoint := 'True'} : Real := 500.0;   // Amount the torq will adjust if increment/decremented. Set on HMI
      OscTorqFwdFtLbs : Real := 5000.0;   // Osc fwd torq setpoint
   END_VAR
   VAR
      OscTorqFwdInc : Bool;   // Increment Torq Fwd
      OscTorqFwdDec : Bool;   // Decrement Torq Fwd
      OscTorqRevInc : Bool;   // Increment Torq Rev
   END_VAR
   VAR RETAIN
      OscTorqRevFtLbs : Real := 5000.0;   // Osc Rev Torq Setpoint
   END_VAR
   VAR
      OscTorqRevDec : Bool;   // Decrement Torq REv
      OscTorqSetPSI : Real;
   END_VAR
   VAR RETAIN
      OscTurnAdj { S7_SetPoint := 'True'} : Real := 0.25;   // Amount the turns will adjust if increment/decremented. Set on HMI
      OscTurnFwd : Real := 1.0;   // Osc Fwd Turns
   END_VAR
   VAR
      OscTurnFwdInc : Bool;   // Increment Turns Fwd
      OscTurnFwdDec : Bool;   // Decrement Turns Fwd
   END_VAR
   VAR RETAIN
      OscTurnRev : Real := 1.0;   // Osc Rev Turns
   END_VAR
   VAR
      OscTurnRevInc : Bool;   // Increment Turns Rev
      OscTurnRevDec : Bool;   // Decrement Turns Rev
      OscTorqFwdLowLimFtlbs : Real;   // Forward torq lower limit based on input and settings
      OscTorqFwdHighLimFtLbs : Real;   // Forward torq high limit based on input and settings
      OscTorqRevLowLimFtlbs : Real;   // Reverse torq lower limit based on input and settings
      OscTorqRevHighLimFtLbs : Real;   // Reverse torq high limit based on input and settings
      OscHomeLowRelDeg : Real;   // Rel Home Position minus 1 count range
      OscHomeLow2RelDeg : Real;   // Rel Home Position minus 2 count range
      OscHomeHighRelDeg : Real;   // Rel Home Position plus 1 count range
      OscHomeHigh2RelDeg : Real;   // Rel Home Position plus 2 count range
      OscPosDeg : Real;   // Degrees of from Home position
      SpareVolts : Real := 0.0;   // Dummy spare Output value used for display
      Spare4MA : Real := 4.0;   // Dummy spare Output value 4ma
      LampTest : Bool;   // Bit used to trigger Console lamp test from HMI
      LampTestLamp_TP { S7_SetPoint := 'True'} : TP_TIME;
      LampTestHorn_TP { S7_SetPoint := 'True'} : TP_TIME;
      ScreenNameInvis { S7_SetPoint := 'True'} : Bool;   // Used to Turn off Screen Name
      ScreenBypassVis : Bool;
      ScreenLampTestVis : Bool;
      HornSilence_TOF { S7_SetPoint := 'True'} : TOF_TIME;
      HornSilenceReset { S7_SetPoint := 'True'} : Bool;   // Horn Silence Bit set on HMI
      Alarms1 : Int;
      Alarms2 : Int;
      Warnings1 : Int;
      Alarms1_To_Unified : Array[0..15] of Bool;
      Alarms2_To_Unified : Array[0..15] of Bool;
      Warnings1_To_Unified : Array[0..15] of Bool;
   END_VAR
   VAR_TEMP
      TempReal : Real;
   END_VAR
   VAR_TEMP   // added for the SCL form of the ladder/FBD networks
      _w1 : Bool;
   END_VAR
BEGIN

REGION Network 1: Oscillator Enable
   // Allow Enable Osciallor Set from HMI if  in Drill, throttle pot set to min and TD stopped, low speed. 
   // HMI Used to Set Enable
   // Reset if Interlocks not met
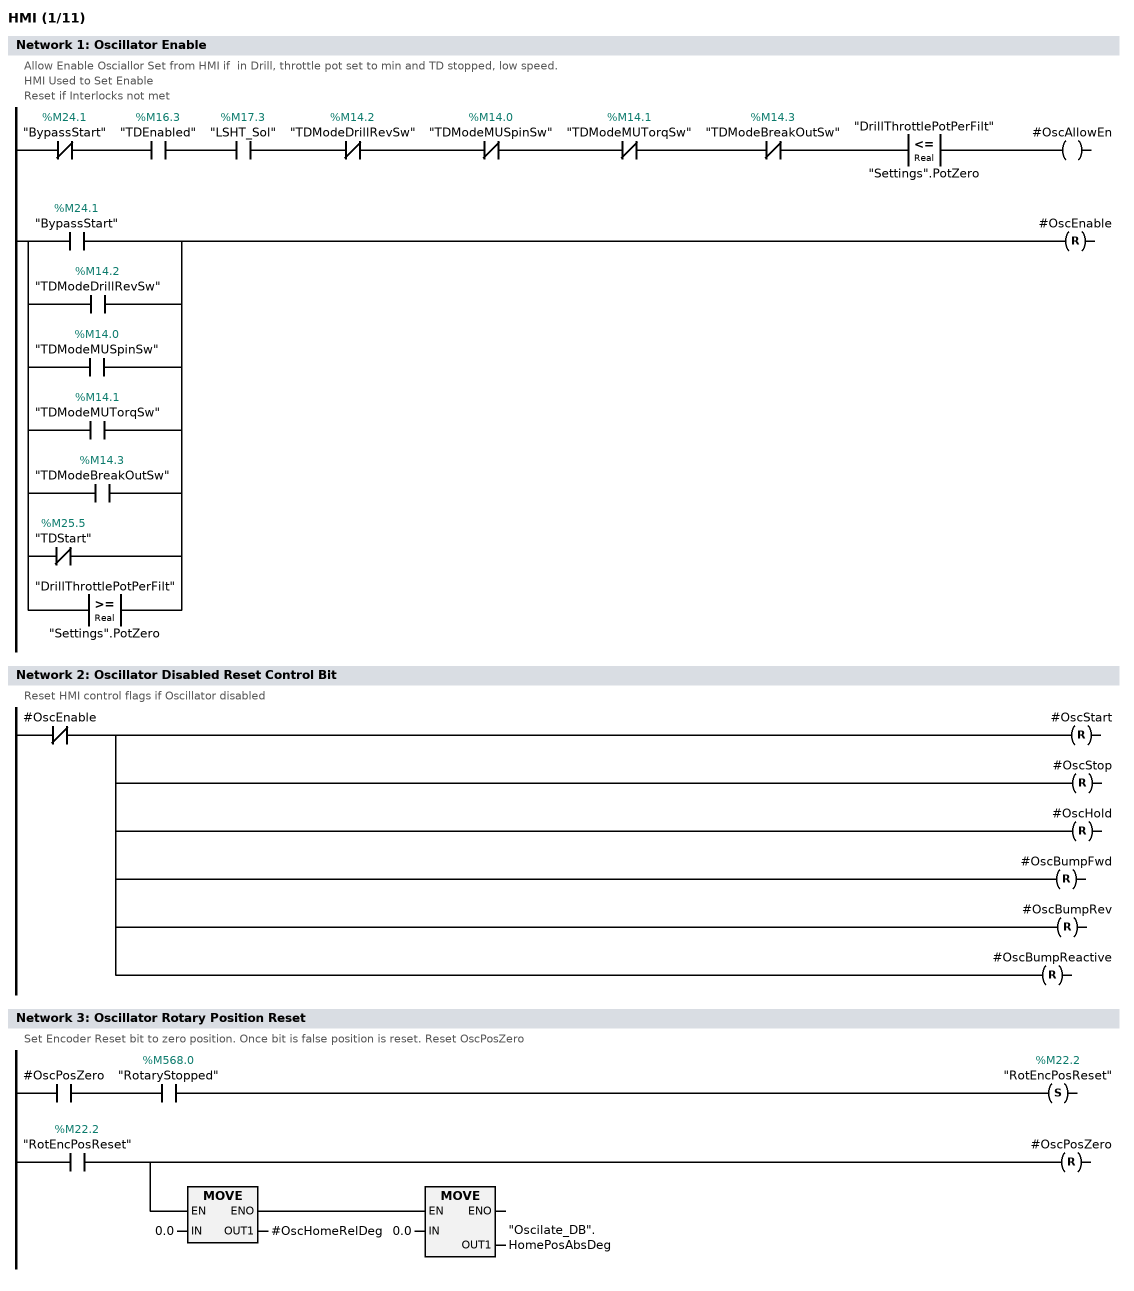
   RUNG wire#powerrail
      I_Contact( "BypassStart" )
      Contact( "TDEnabled" )
      Contact( "LSHT_Sol" )
      I_Contact( "TDModeDrillRevSw" )
      I_Contact( "TDModeMUSpinSw" )
      I_Contact( "TDModeMUTorqSw" )
      I_Contact( "TDModeBreakOutSw" )
      { S7_Templates := "SrcType := Real" } LE_Contact(in1 := "DrillThrottlePotPerFilt", in2 := "Settings".PotZero)
      Coil( #OscAllowEn )
   END_RUNG
   RUNG wire#powerrail
      Contact( "BypassStart" )
      wire#w1
      R_Coil( #OscEnable )
   END_RUNG
   RUNG wire#powerrail
      Contact( "TDModeDrillRevSw" )
   END_RUNG wire#w1
   RUNG wire#powerrail
      Contact( "TDModeMUSpinSw" )
   END_RUNG wire#w1
   RUNG wire#powerrail
      Contact( "TDModeMUTorqSw" )
   END_RUNG wire#w1
   RUNG wire#powerrail
      Contact( "TDModeBreakOutSw" )
   END_RUNG wire#w1
   RUNG wire#powerrail
      I_Contact( "TDStart" )
   END_RUNG wire#w1
   RUNG wire#powerrail
      { S7_Templates := "SrcType := Real" } GE_Contact(in1 := "DrillThrottlePotPerFilt", in2 := "Settings".PotZero)
   END_RUNG wire#w1
   // the same network as SCL:
   #OscAllowEn := NOT "BypassStart" AND "TDEnabled" AND "LSHT_Sol" AND NOT "TDModeDrillRevSw" AND NOT "TDModeMUSpinSw" AND NOT "TDModeMUTorqSw" AND NOT "TDModeBreakOutSw" AND ("DrillThrottlePotPerFilt" <= "Settings".PotZero);
   IF "BypassStart" OR "TDModeDrillRevSw" OR "TDModeMUSpinSw" OR "TDModeMUTorqSw" OR "TDModeBreakOutSw" OR NOT "TDStart" OR ("DrillThrottlePotPerFilt" >= "Settings".PotZero) THEN
       #OscEnable := FALSE;
   END_IF;
END_REGION

REGION Network 2: Oscillator Disabled Reset Control Bit
   // Reset HMI control flags if Oscillator disabled
   RUNG wire#powerrail
      I_Contact( #OscEnable )
      wire#w1
      R_Coil( #OscStart )
   END_RUNG
   RUNG wire#w1
      R_Coil( #OscStop )
   END_RUNG
   RUNG wire#w1
      R_Coil( #OscHold )
   END_RUNG
   RUNG wire#w1
      R_Coil( #OscBumpFwd )
   END_RUNG
   RUNG wire#w1
      R_Coil( #OscBumpRev )
   END_RUNG
   RUNG wire#w1
      R_Coil( #OscBumpReactive )
   END_RUNG
   // the same network as SCL:
   IF NOT #OscEnable THEN
       #OscStart := FALSE;
       #OscStop := FALSE;
       #OscHold := FALSE;
       #OscBumpFwd := FALSE;
       #OscBumpRev := FALSE;
       #OscBumpReactive := FALSE;
   END_IF;
END_REGION

REGION Network 3: Oscillator Rotary Position Reset
   // Set Encoder Reset bit to zero position. Once bit is false position is reset. Reset OscPosZero
   RUNG wire#powerrail
      Contact( #OscPosZero )
      Contact( "RotaryStopped" )
      S_Coil( "RotEncPosReset" )
   END_RUNG
   RUNG wire#powerrail
      Contact( "RotEncPosReset" )
      wire#w1
      R_Coil( #OscPosZero )
   END_RUNG
   RUNG wire#w1
      Move(in := 0.0, out1 => #OscHomeRelDeg)
      Move(in := 0.0, out1 => "Oscilate_DB".HomePosAbsDeg)
   END_RUNG
   // the same network as SCL:
   IF #OscPosZero AND "RotaryStopped" THEN "RotEncPosReset" := TRUE; END_IF;
   IF "RotEncPosReset" THEN
       #OscPosZero := FALSE;
       #OscHomeRelDeg := 0.0;
       "Oscilate_DB".HomePosAbsDeg := 0.0;
   END_IF;
END_REGION

REGION Network 4: Oscillator Position
   // Determine Oscillation position based on home position and actual absolute position
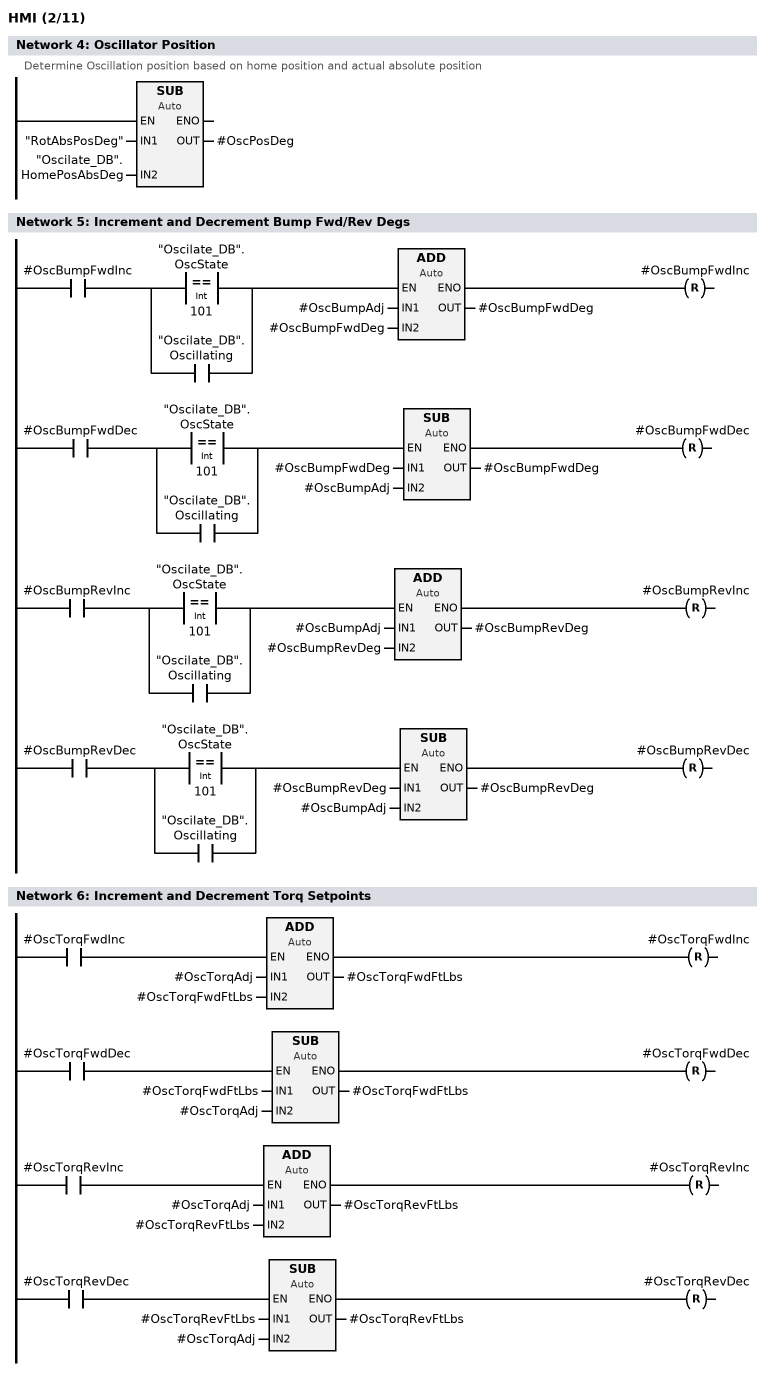
   RUNG wire#powerrail
      Sub(in1 := "RotAbsPosDeg", in2 := "Oscilate_DB".HomePosAbsDeg, out => #OscPosDeg)
   END_RUNG
   // the same network as SCL:
   #OscPosDeg := "RotAbsPosDeg" - "Oscilate_DB".HomePosAbsDeg;
END_REGION

REGION Network 5: Increment and Decrement Bump Fwd/Rev Degs
   RUNG wire#powerrail
      Contact( #OscBumpFwdInc )
      wire#w1
      { S7_Templates := "SrcType := Int" } EQ_Contact(in1 := "Oscilate_DB".OscState, in2 := 101)
      wire#w2
      Add(in1 := #OscBumpAdj, in2 := #OscBumpFwdDeg, out => #OscBumpFwdDeg)
      R_Coil( #OscBumpFwdInc )
   END_RUNG
   RUNG wire#w1
      Contact( "Oscilate_DB".Oscillating )
   END_RUNG wire#w2
   RUNG wire#powerrail
      Contact( #OscBumpFwdDec )
      wire#w3
      { S7_Templates := "SrcType := Int" } EQ_Contact(in1 := "Oscilate_DB".OscState, in2 := 101)
      wire#w4
      Sub(in1 := #OscBumpFwdDeg, in2 := #OscBumpAdj, out => #OscBumpFwdDeg)
      R_Coil( #OscBumpFwdDec )
   END_RUNG
   RUNG wire#w3
      Contact( "Oscilate_DB".Oscillating )
   END_RUNG wire#w4
   RUNG wire#powerrail
      Contact( #OscBumpRevInc )
      wire#w5
      { S7_Templates := "SrcType := Int" } EQ_Contact(in1 := "Oscilate_DB".OscState, in2 := 101)
      wire#w6
      Add(in1 := #OscBumpAdj, in2 := #OscBumpRevDeg, out => #OscBumpRevDeg)
      R_Coil( #OscBumpRevInc )
   END_RUNG
   RUNG wire#w5
      Contact( "Oscilate_DB".Oscillating )
   END_RUNG wire#w6
   RUNG wire#powerrail
      Contact( #OscBumpRevDec )
      wire#w7
      { S7_Templates := "SrcType := Int" } EQ_Contact(in1 := "Oscilate_DB".OscState, in2 := 101)
      wire#w8
      Sub(in1 := #OscBumpRevDeg, in2 := #OscBumpAdj, out => #OscBumpRevDeg)
      R_Coil( #OscBumpRevDec )
   END_RUNG
   RUNG wire#w7
      Contact( "Oscilate_DB".Oscillating )
   END_RUNG wire#w8
   // the same network as SCL:
   IF #OscBumpFwdInc AND (("Oscilate_DB".OscState = 101) OR "Oscilate_DB".Oscillating) THEN
       #OscBumpFwdDeg := #OscBumpAdj + #OscBumpFwdDeg;
       #OscBumpFwdInc := FALSE;
   END_IF;
   IF #OscBumpFwdDec AND (("Oscilate_DB".OscState = 101) OR "Oscilate_DB".Oscillating) THEN
       #OscBumpFwdDeg := #OscBumpFwdDeg - #OscBumpAdj;
       #OscBumpFwdDec := FALSE;
   END_IF;
   IF #OscBumpRevInc AND (("Oscilate_DB".OscState = 101) OR "Oscilate_DB".Oscillating) THEN
       #OscBumpRevDeg := #OscBumpAdj + #OscBumpRevDeg;
       #OscBumpRevInc := FALSE;
   END_IF;
   IF #OscBumpRevDec AND (("Oscilate_DB".OscState = 101) OR "Oscilate_DB".Oscillating) THEN
       #OscBumpRevDeg := #OscBumpRevDeg - #OscBumpAdj;
       #OscBumpRevDec := FALSE;
   END_IF;
END_REGION

REGION Network 6: Increment and Decrement Torq Setpoints
   RUNG wire#powerrail
      Contact( #OscTorqFwdInc )
      Add(in1 := #OscTorqAdj, in2 := #OscTorqFwdFtLbs, out => #OscTorqFwdFtLbs)
      R_Coil( #OscTorqFwdInc )
   END_RUNG
   RUNG wire#powerrail
      Contact( #OscTorqFwdDec )
      Sub(in1 := #OscTorqFwdFtLbs, in2 := #OscTorqAdj, out => #OscTorqFwdFtLbs)
      R_Coil( #OscTorqFwdDec )
   END_RUNG
   RUNG wire#powerrail
      Contact( #OscTorqRevInc )
      Add(in1 := #OscTorqAdj, in2 := #OscTorqRevFtLbs, out => #OscTorqRevFtLbs)
      R_Coil( #OscTorqRevInc )
   END_RUNG
   RUNG wire#powerrail
      Contact( #OscTorqRevDec )
      Sub(in1 := #OscTorqRevFtLbs, in2 := #OscTorqAdj, out => #OscTorqRevFtLbs)
      R_Coil( #OscTorqRevDec )
   END_RUNG
   // the same network as SCL:
   IF #OscTorqFwdInc THEN
       #OscTorqFwdFtLbs := #OscTorqAdj + #OscTorqFwdFtLbs;
       #OscTorqFwdInc := FALSE;
   END_IF;
   IF #OscTorqFwdDec THEN
       #OscTorqFwdFtLbs := #OscTorqFwdFtLbs - #OscTorqAdj;
       #OscTorqFwdDec := FALSE;
   END_IF;
   IF #OscTorqRevInc THEN
       #OscTorqRevFtLbs := #OscTorqAdj + #OscTorqRevFtLbs;
       #OscTorqRevInc := FALSE;
   END_IF;
   IF #OscTorqRevDec THEN
       #OscTorqRevFtLbs := #OscTorqRevFtLbs - #OscTorqAdj;
       #OscTorqRevDec := FALSE;
   END_IF;
END_REGION

REGION Network 7: Increment and Decrement Turns
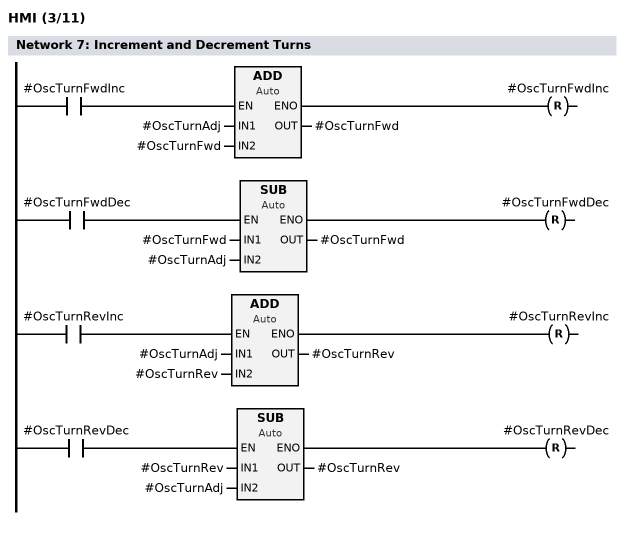
   RUNG wire#powerrail
      Contact( #OscTurnFwdInc )
      Add(in1 := #OscTurnAdj, in2 := #OscTurnFwd, out => #OscTurnFwd)
      R_Coil( #OscTurnFwdInc )
   END_RUNG
   RUNG wire#powerrail
      Contact( #OscTurnFwdDec )
      Sub(in1 := #OscTurnFwd, in2 := #OscTurnAdj, out => #OscTurnFwd)
      R_Coil( #OscTurnFwdDec )
   END_RUNG
   RUNG wire#powerrail
      Contact( #OscTurnRevInc )
      Add(in1 := #OscTurnAdj, in2 := #OscTurnRev, out => #OscTurnRev)
      R_Coil( #OscTurnRevInc )
   END_RUNG
   RUNG wire#powerrail
      Contact( #OscTurnRevDec )
      Sub(in1 := #OscTurnRev, in2 := #OscTurnAdj, out => #OscTurnRev)
      R_Coil( #OscTurnRevDec )
   END_RUNG
   // the same network as SCL:
   IF #OscTurnFwdInc THEN
       #OscTurnFwd := #OscTurnAdj + #OscTurnFwd;
       #OscTurnFwdInc := FALSE;
   END_IF;
   IF #OscTurnFwdDec THEN
       #OscTurnFwd := #OscTurnFwd - #OscTurnAdj;
       #OscTurnFwdDec := FALSE;
   END_IF;
   IF #OscTurnRevInc THEN
       #OscTurnRev := #OscTurnAdj + #OscTurnRev;
       #OscTurnRevInc := FALSE;
   END_IF;
   IF #OscTurnRevDec THEN
       #OscTurnRev := #OscTurnRev - #OscTurnAdj;
       #OscTurnRevDec := FALSE;
   END_IF;
END_REGION

REGION Network 8: Oscillator Input Limits Checks
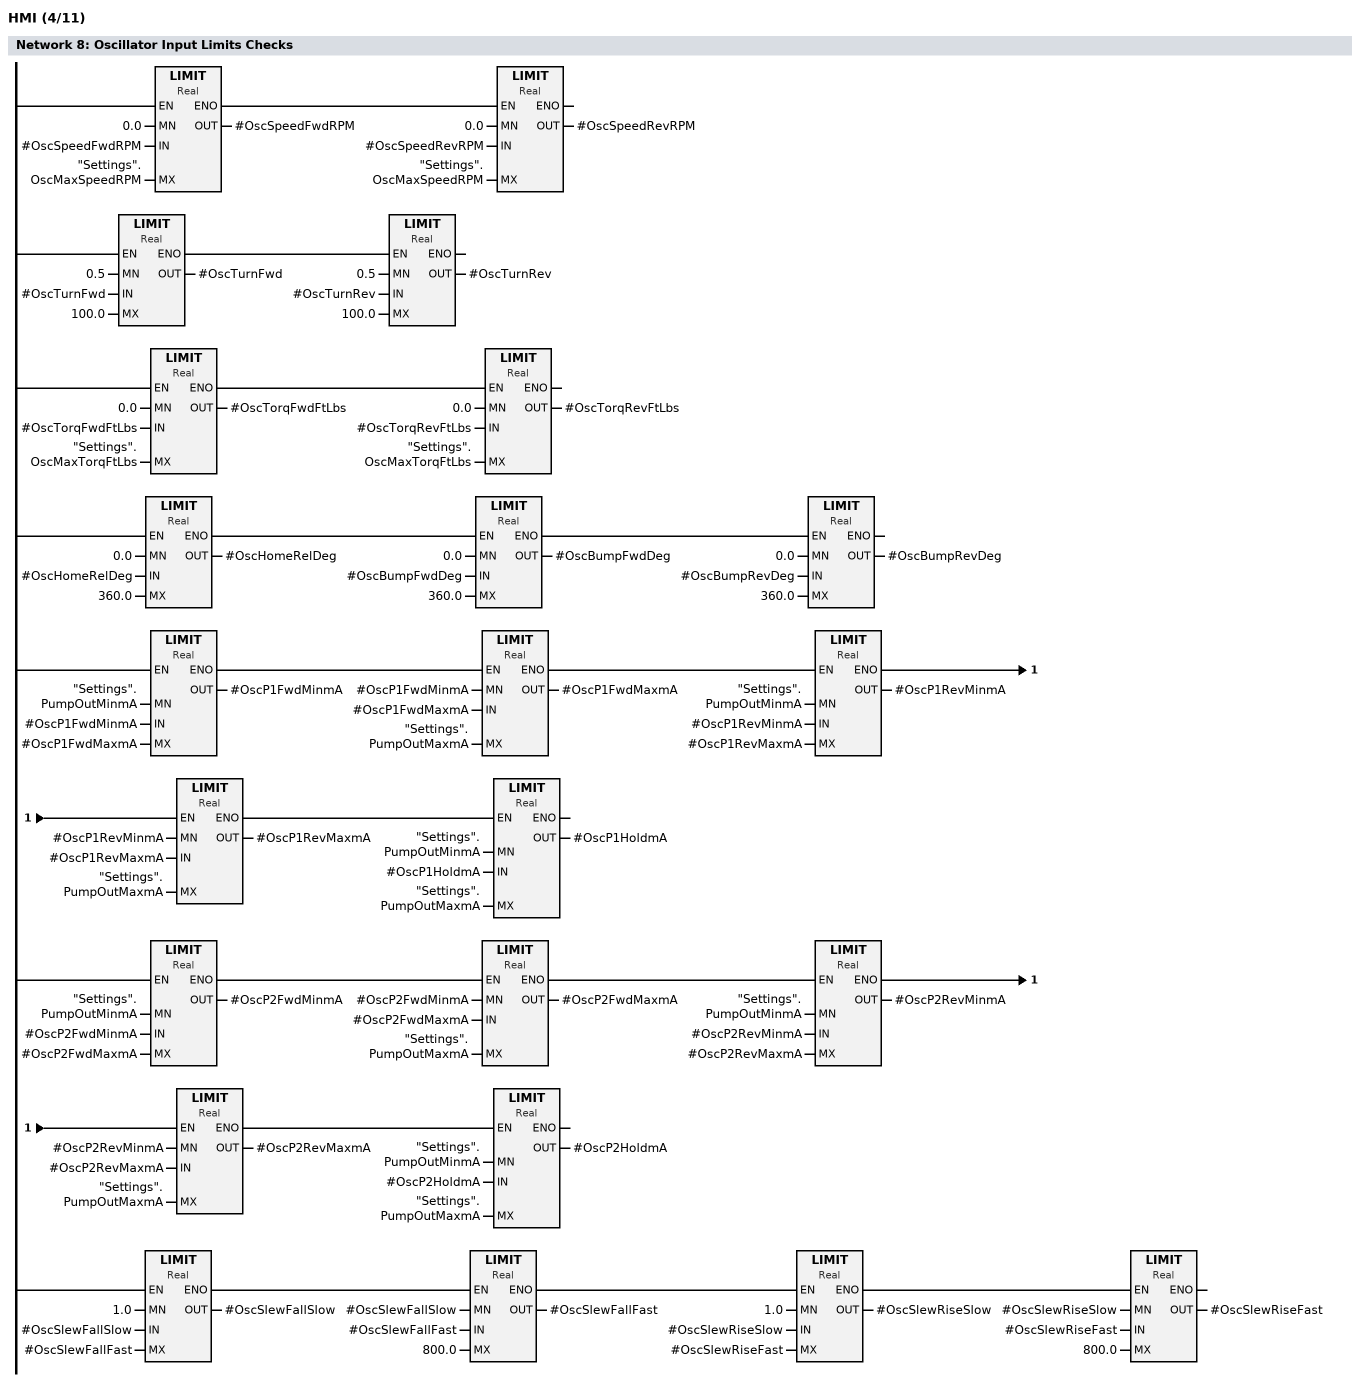
   RUNG wire#powerrail
      { S7_Templates := "value_type := Real" } Limit(mn := 0.0, in := #OscSpeedFwdRPM, mx := "Settings".OscMaxSpeedRPM, out => #OscSpeedFwdRPM)
      { S7_Templates := "value_type := Real" } Limit(mn := 0.0, in := #OscSpeedRevRPM, mx := "Settings".OscMaxSpeedRPM, out => #OscSpeedRevRPM)
   END_RUNG
   RUNG wire#powerrail
      { S7_Templates := "value_type := Real" } Limit(mn := 0.5, in := #OscTurnFwd, mx := 100.0, out => #OscTurnFwd)
      { S7_Templates := "value_type := Real" } Limit(mn := 0.5, in := #OscTurnRev, mx := 100.0, out => #OscTurnRev)
   END_RUNG
   RUNG wire#powerrail
      { S7_Templates := "value_type := Real" } Limit(mn := 0.0, in := #OscTorqFwdFtLbs, mx := "Settings".OscMaxTorqFtLbs, out => #OscTorqFwdFtLbs)
      { S7_Templates := "value_type := Real" } Limit(mn := 0.0, in := #OscTorqRevFtLbs, mx := "Settings".OscMaxTorqFtLbs, out => #OscTorqRevFtLbs)
   END_RUNG
   RUNG wire#powerrail
      { S7_Templates := "value_type := Real" } Limit(mn := 0.0, in := #OscHomeRelDeg, mx := 360.0, out => #OscHomeRelDeg)
      { S7_Templates := "value_type := Real" } Limit(mn := 0.0, in := #OscBumpFwdDeg, mx := 360.0, out => #OscBumpFwdDeg)
      { S7_Templates := "value_type := Real" } Limit(mn := 0.0, in := #OscBumpRevDeg, mx := 360.0, out => #OscBumpRevDeg)
   END_RUNG
   RUNG wire#powerrail
      { S7_Templates := "value_type := Real" } Limit(mn := "Settings".PumpOutMinmA, in := #OscP1FwdMinmA, mx := #OscP1FwdMaxmA, out => #OscP1FwdMinmA)
      { S7_Templates := "value_type := Real" } Limit(mn := #OscP1FwdMinmA, in := #OscP1FwdMaxmA, mx := "Settings".PumpOutMaxmA, out => #OscP1FwdMaxmA)
      { S7_Templates := "value_type := Real" } Limit(mn := "Settings".PumpOutMinmA, in := #OscP1RevMinmA, mx := #OscP1RevMaxmA, out => #OscP1RevMinmA)
      { S7_Templates := "value_type := Real" } Limit(mn := #OscP1RevMinmA, in := #OscP1RevMaxmA, mx := "Settings".PumpOutMaxmA, out => #OscP1RevMaxmA)
      { S7_Templates := "value_type := Real" } Limit(mn := "Settings".PumpOutMinmA, in := #OscP1HoldmA, mx := "Settings".PumpOutMaxmA, out => #OscP1HoldmA)
   END_RUNG
   RUNG wire#powerrail
      { S7_Templates := "value_type := Real" } Limit(mn := "Settings".PumpOutMinmA, in := #OscP2FwdMinmA, mx := #OscP2FwdMaxmA, out => #OscP2FwdMinmA)
      { S7_Templates := "value_type := Real" } Limit(mn := #OscP2FwdMinmA, in := #OscP2FwdMaxmA, mx := "Settings".PumpOutMaxmA, out => #OscP2FwdMaxmA)
      { S7_Templates := "value_type := Real" } Limit(mn := "Settings".PumpOutMinmA, in := #OscP2RevMinmA, mx := #OscP2RevMaxmA, out => #OscP2RevMinmA)
      { S7_Templates := "value_type := Real" } Limit(mn := #OscP2RevMinmA, in := #OscP2RevMaxmA, mx := "Settings".PumpOutMaxmA, out => #OscP2RevMaxmA)
      { S7_Templates := "value_type := Real" } Limit(mn := "Settings".PumpOutMinmA, in := #OscP2HoldmA, mx := "Settings".PumpOutMaxmA, out => #OscP2HoldmA)
   END_RUNG
   RUNG wire#powerrail
      { S7_Templates := "value_type := Real" } Limit(mn := 1.0, in := #OscSlewFallSlow, mx := #OscSlewFallFast, out => #OscSlewFallSlow)
      { S7_Templates := "value_type := Real" } Limit(mn := #OscSlewFallSlow, in := #OscSlewFallFast, mx := 800.0, out => #OscSlewFallFast)
      { S7_Templates := "value_type := Real" } Limit(mn := 1.0, in := #OscSlewRiseSlow, mx := #OscSlewRiseFast, out => #OscSlewRiseSlow)
      { S7_Templates := "value_type := Real" } Limit(mn := #OscSlewRiseSlow, in := #OscSlewRiseFast, mx := 800.0, out => #OscSlewRiseFast)
   END_RUNG
   // the same network as SCL:
   #OscSpeedFwdRPM := LIMIT(MN := 0.0, IN := #OscSpeedFwdRPM, MX := "Settings".OscMaxSpeedRPM);
   #OscSpeedRevRPM := LIMIT(MN := 0.0, IN := #OscSpeedRevRPM, MX := "Settings".OscMaxSpeedRPM);
   #OscTurnFwd := LIMIT(MN := 0.5, IN := #OscTurnFwd, MX := 100.0);
   #OscTurnRev := LIMIT(MN := 0.5, IN := #OscTurnRev, MX := 100.0);
   #OscTorqFwdFtLbs := LIMIT(MN := 0.0, IN := #OscTorqFwdFtLbs, MX := "Settings".OscMaxTorqFtLbs);
   #OscTorqRevFtLbs := LIMIT(MN := 0.0, IN := #OscTorqRevFtLbs, MX := "Settings".OscMaxTorqFtLbs);
   #OscHomeRelDeg := LIMIT(MN := 0.0, IN := #OscHomeRelDeg, MX := 360.0);
   #OscBumpFwdDeg := LIMIT(MN := 0.0, IN := #OscBumpFwdDeg, MX := 360.0);
   #OscBumpRevDeg := LIMIT(MN := 0.0, IN := #OscBumpRevDeg, MX := 360.0);
   #OscP1FwdMinmA := LIMIT(MN := "Settings".PumpOutMinmA, IN := #OscP1FwdMinmA, MX := #OscP1FwdMaxmA);
   #OscP1FwdMaxmA := LIMIT(MN := #OscP1FwdMinmA, IN := #OscP1FwdMaxmA, MX := "Settings".PumpOutMaxmA);
   #OscP1RevMinmA := LIMIT(MN := "Settings".PumpOutMinmA, IN := #OscP1RevMinmA, MX := #OscP1RevMaxmA);
   #OscP1RevMaxmA := LIMIT(MN := #OscP1RevMinmA, IN := #OscP1RevMaxmA, MX := "Settings".PumpOutMaxmA);
   #OscP1HoldmA := LIMIT(MN := "Settings".PumpOutMinmA, IN := #OscP1HoldmA, MX := "Settings".PumpOutMaxmA);
   #OscP2FwdMinmA := LIMIT(MN := "Settings".PumpOutMinmA, IN := #OscP2FwdMinmA, MX := #OscP2FwdMaxmA);
   #OscP2FwdMaxmA := LIMIT(MN := #OscP2FwdMinmA, IN := #OscP2FwdMaxmA, MX := "Settings".PumpOutMaxmA);
   #OscP2RevMinmA := LIMIT(MN := "Settings".PumpOutMinmA, IN := #OscP2RevMinmA, MX := #OscP2RevMaxmA);
   #OscP2RevMaxmA := LIMIT(MN := #OscP2RevMinmA, IN := #OscP2RevMaxmA, MX := "Settings".PumpOutMaxmA);
   #OscP2HoldmA := LIMIT(MN := "Settings".PumpOutMinmA, IN := #OscP2HoldmA, MX := "Settings".PumpOutMaxmA);
   #OscSlewFallSlow := LIMIT(MN := 1.0, IN := #OscSlewFallSlow, MX := #OscSlewFallFast);
   #OscSlewFallFast := LIMIT(MN := #OscSlewFallSlow, IN := #OscSlewFallFast, MX := 800.0);
   #OscSlewRiseSlow := LIMIT(MN := 1.0, IN := #OscSlewRiseSlow, MX := #OscSlewRiseFast);
   #OscSlewRiseFast := LIMIT(MN := #OscSlewRiseSlow, IN := #OscSlewRiseFast, MX := 800.0);
END_REGION

REGION Network 9: Calculate Torq Setpoint
   // Only Fwd Torq is used to set torq
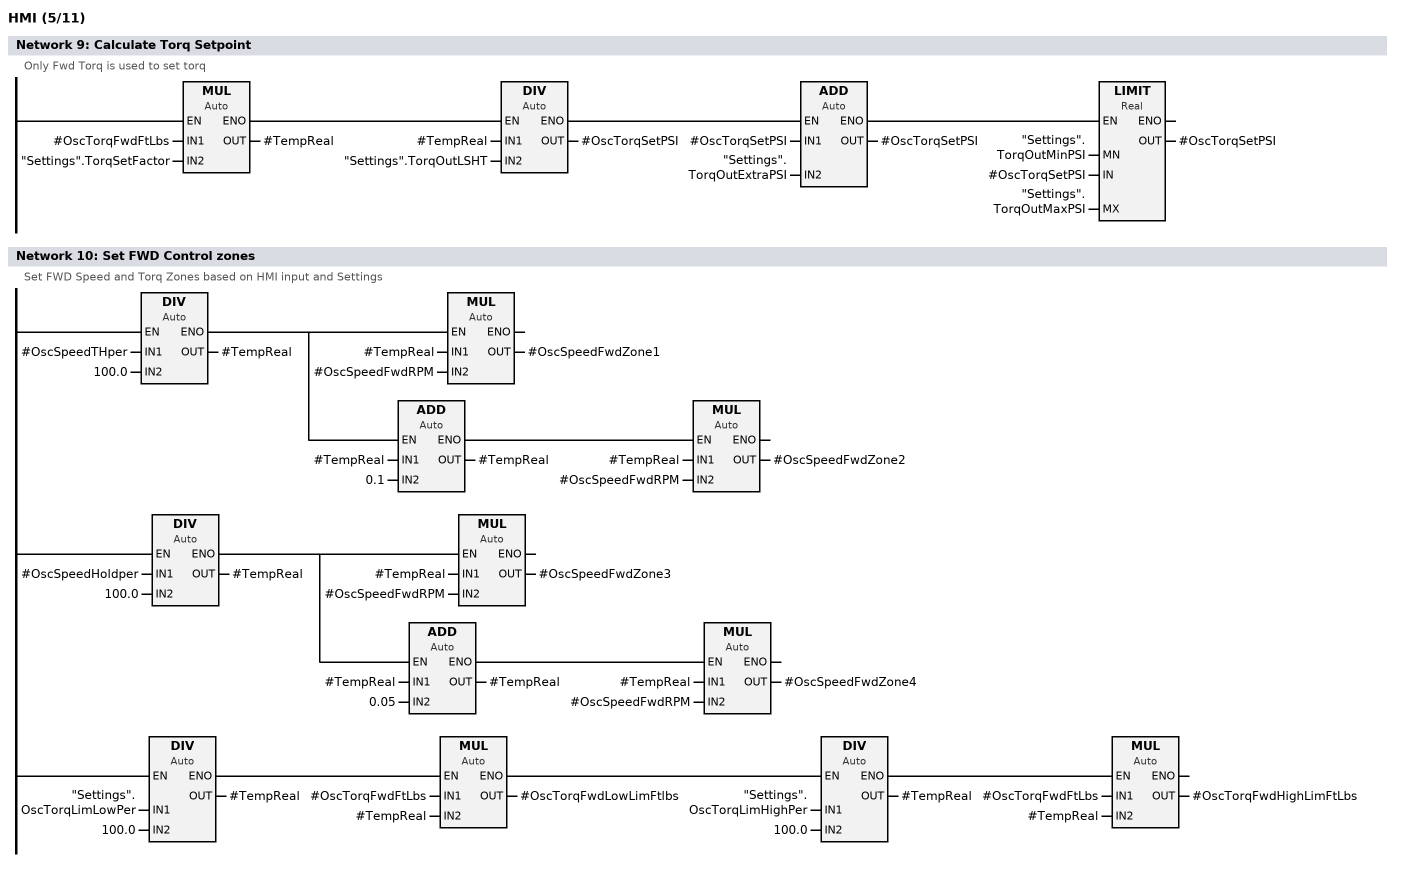
   RUNG wire#powerrail
      Mul(in1 := #OscTorqFwdFtLbs, in2 := "Settings".TorqSetFactor, out => #TempReal)
      Div(in1 := #TempReal, in2 := "Settings".TorqOutLSHT, out => #OscTorqSetPSI)
      Add(in1 := #OscTorqSetPSI, in2 := "Settings".TorqOutExtraPSI, out => #OscTorqSetPSI)
      { S7_Templates := "value_type := Real" } Limit(mn := "Settings".TorqOutMinPSI, in := #OscTorqSetPSI, mx := "Settings".TorqOutMaxPSI, out => #OscTorqSetPSI)
   END_RUNG
   // the same network as SCL:
   #TempReal := #OscTorqFwdFtLbs * "Settings".TorqSetFactor;
   #OscTorqSetPSI := #TempReal / "Settings".TorqOutLSHT;
   #OscTorqSetPSI := #OscTorqSetPSI + "Settings".TorqOutExtraPSI;
   #OscTorqSetPSI := LIMIT(MN := "Settings".TorqOutMinPSI, IN := #OscTorqSetPSI, MX := "Settings".TorqOutMaxPSI);
END_REGION

REGION Network 10: Set FWD Control zones
   // Set FWD Speed and Torq Zones based on HMI input and Settings
   RUNG wire#powerrail
      Div(in1 := #OscSpeedTHper, in2 := 100.0, out => #TempReal)
      wire#w1
      Mul(in1 := #TempReal, in2 := #OscSpeedFwdRPM, out => #OscSpeedFwdZone1)
   END_RUNG
   RUNG wire#w1
      Add(in1 := #TempReal, in2 := 0.1, out => #TempReal)
      Mul(in1 := #TempReal, in2 := #OscSpeedFwdRPM, out => #OscSpeedFwdZone2)
   END_RUNG
   RUNG wire#powerrail
      Div(in1 := #OscSpeedHoldper, in2 := 100.0, out => #TempReal)
      wire#w2
      Mul(in1 := #TempReal, in2 := #OscSpeedFwdRPM, out => #OscSpeedFwdZone3)
   END_RUNG
   RUNG wire#w2
      Add(in1 := #TempReal, in2 := 0.05, out => #TempReal)
      Mul(in1 := #TempReal, in2 := #OscSpeedFwdRPM, out => #OscSpeedFwdZone4)
   END_RUNG
   RUNG wire#powerrail
      Div(in1 := "Settings".OscTorqLimLowPer, in2 := 100.0, out => #TempReal)
      Mul(in1 := #OscTorqFwdFtLbs, in2 := #TempReal, out => #OscTorqFwdLowLimFtlbs)
      Div(in1 := "Settings".OscTorqLimHighPer, in2 := 100.0, out => #TempReal)
      Mul(in1 := #OscTorqFwdFtLbs, in2 := #TempReal, out => #OscTorqFwdHighLimFtLbs)
   END_RUNG
   // the same network as SCL:
   #TempReal := #OscSpeedTHper / 100.0;
   #OscSpeedFwdZone1 := #TempReal * #OscSpeedFwdRPM;
   #TempReal := #TempReal + 0.1;
   #OscSpeedFwdZone2 := #TempReal * #OscSpeedFwdRPM;
   #TempReal := #OscSpeedHoldper / 100.0;
   #OscSpeedFwdZone3 := #TempReal * #OscSpeedFwdRPM;
   #TempReal := #TempReal + 0.05;
   #OscSpeedFwdZone4 := #TempReal * #OscSpeedFwdRPM;
   #TempReal := "Settings".OscTorqLimLowPer / 100.0;
   #OscTorqFwdLowLimFtlbs := #OscTorqFwdFtLbs * #TempReal;
   #TempReal := "Settings".OscTorqLimHighPer / 100.0;
   #OscTorqFwdHighLimFtLbs := #OscTorqFwdFtLbs * #TempReal;
END_REGION

REGION Network 11: Set Rev Controls zones
   // Set Rev Speed and Torq Zones based on HMI input and Settings
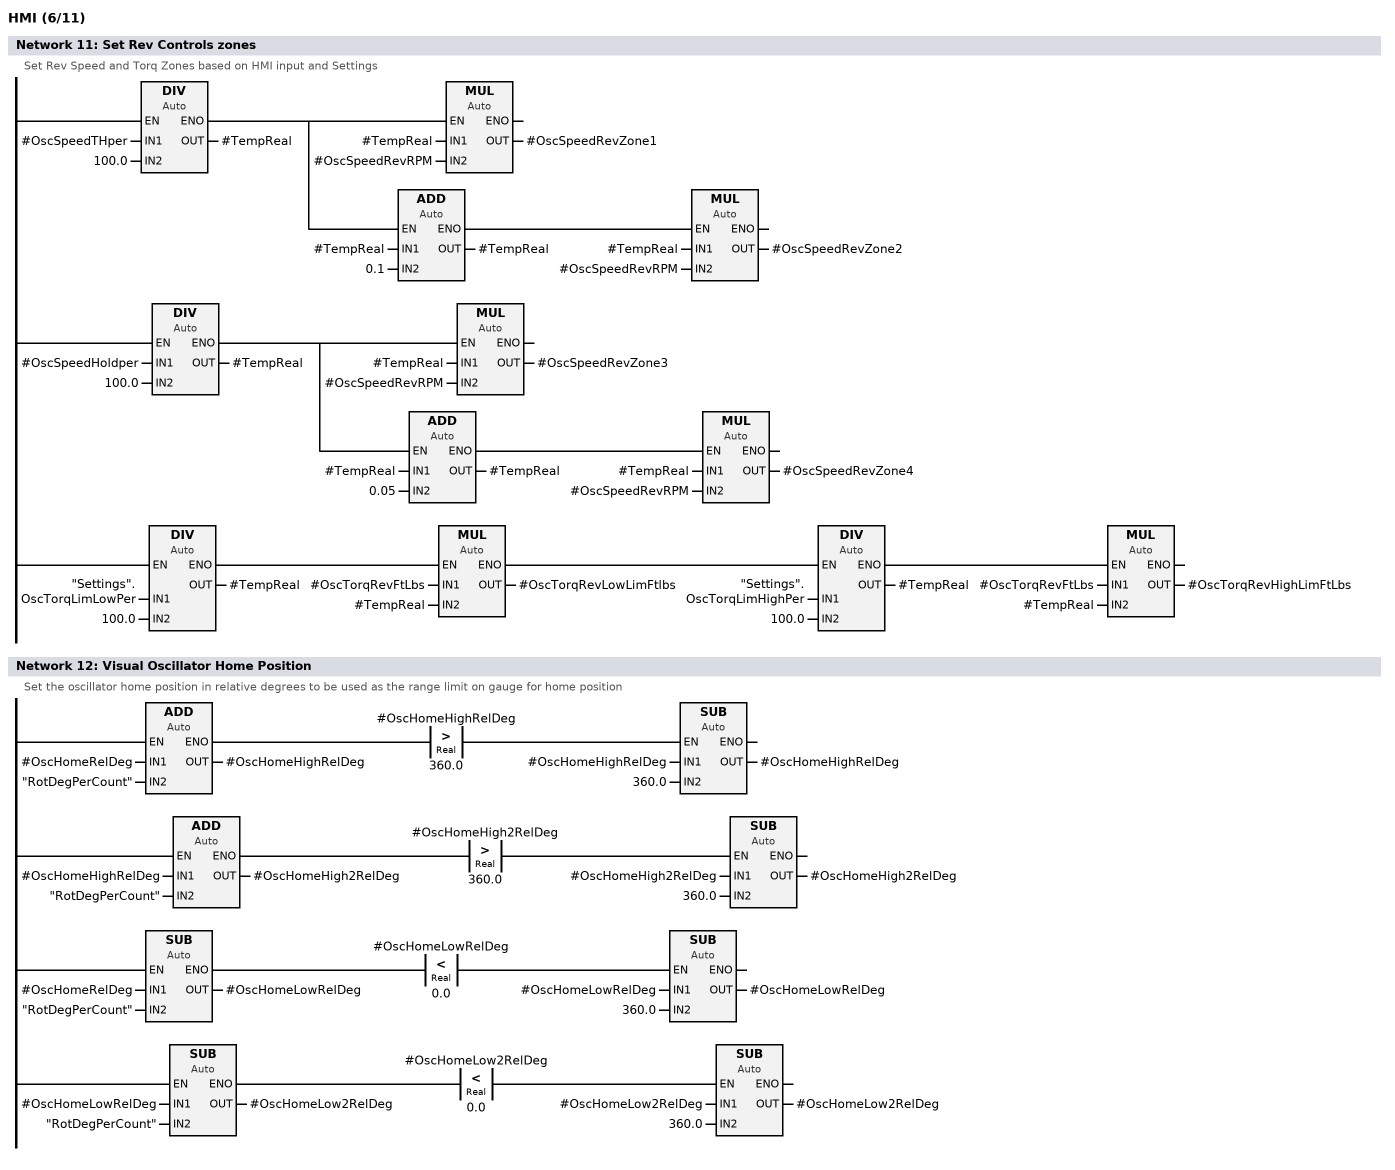
   RUNG wire#powerrail
      Div(in1 := #OscSpeedTHper, in2 := 100.0, out => #TempReal)
      wire#w1
      Mul(in1 := #TempReal, in2 := #OscSpeedRevRPM, out => #OscSpeedRevZone1)
   END_RUNG
   RUNG wire#w1
      Add(in1 := #TempReal, in2 := 0.1, out => #TempReal)
      Mul(in1 := #TempReal, in2 := #OscSpeedRevRPM, out => #OscSpeedRevZone2)
   END_RUNG
   RUNG wire#powerrail
      Div(in1 := #OscSpeedHoldper, in2 := 100.0, out => #TempReal)
      wire#w2
      Mul(in1 := #TempReal, in2 := #OscSpeedRevRPM, out => #OscSpeedRevZone3)
   END_RUNG
   RUNG wire#w2
      Add(in1 := #TempReal, in2 := 0.05, out => #TempReal)
      Mul(in1 := #TempReal, in2 := #OscSpeedRevRPM, out => #OscSpeedRevZone4)
   END_RUNG
   RUNG wire#powerrail
      Div(in1 := "Settings".OscTorqLimLowPer, in2 := 100.0, out => #TempReal)
      Mul(in1 := #OscTorqRevFtLbs, in2 := #TempReal, out => #OscTorqRevLowLimFtlbs)
      Div(in1 := "Settings".OscTorqLimHighPer, in2 := 100.0, out => #TempReal)
      Mul(in1 := #OscTorqRevFtLbs, in2 := #TempReal, out => #OscTorqRevHighLimFtLbs)
   END_RUNG
   // the same network as SCL:
   #TempReal := #OscSpeedTHper / 100.0;
   #OscSpeedRevZone1 := #TempReal * #OscSpeedRevRPM;
   #TempReal := #TempReal + 0.1;
   #OscSpeedRevZone2 := #TempReal * #OscSpeedRevRPM;
   #TempReal := #OscSpeedHoldper / 100.0;
   #OscSpeedRevZone3 := #TempReal * #OscSpeedRevRPM;
   #TempReal := #TempReal + 0.05;
   #OscSpeedRevZone4 := #TempReal * #OscSpeedRevRPM;
   #TempReal := "Settings".OscTorqLimLowPer / 100.0;
   #OscTorqRevLowLimFtlbs := #OscTorqRevFtLbs * #TempReal;
   #TempReal := "Settings".OscTorqLimHighPer / 100.0;
   #OscTorqRevHighLimFtLbs := #OscTorqRevFtLbs * #TempReal;
END_REGION

REGION Network 12: Visual Oscillator Home Position
   // Set the oscillator home position in relative degrees to be used as the range limit on gauge for home position
   RUNG wire#powerrail
      Add(in1 := #OscHomeRelDeg, in2 := "RotDegPerCount", out => #OscHomeHighRelDeg)
      { S7_Templates := "SrcType := Real" } GT_Contact(in1 := #OscHomeHighRelDeg, in2 := 360.0)
      Sub(in1 := #OscHomeHighRelDeg, in2 := 360.0, out => #OscHomeHighRelDeg)
   END_RUNG
   RUNG wire#powerrail
      Add(in1 := #OscHomeHighRelDeg, in2 := "RotDegPerCount", out => #OscHomeHigh2RelDeg)
      { S7_Templates := "SrcType := Real" } GT_Contact(in1 := #OscHomeHigh2RelDeg, in2 := 360.0)
      Sub(in1 := #OscHomeHigh2RelDeg, in2 := 360.0, out => #OscHomeHigh2RelDeg)
   END_RUNG
   RUNG wire#powerrail
      Sub(in1 := #OscHomeRelDeg, in2 := "RotDegPerCount", out => #OscHomeLowRelDeg)
      { S7_Templates := "SrcType := Real" } LT_Contact(in1 := #OscHomeLowRelDeg, in2 := 0.0)
      Sub(in1 := #OscHomeLowRelDeg, in2 := 360.0, out => #OscHomeLowRelDeg)
   END_RUNG
   RUNG wire#powerrail
      Sub(in1 := #OscHomeLowRelDeg, in2 := "RotDegPerCount", out => #OscHomeLow2RelDeg)
      { S7_Templates := "SrcType := Real" } LT_Contact(in1 := #OscHomeLow2RelDeg, in2 := 0.0)
      Sub(in1 := #OscHomeLow2RelDeg, in2 := 360.0, out => #OscHomeLow2RelDeg)
   END_RUNG
   // the same network as SCL:
   #OscHomeHighRelDeg := #OscHomeRelDeg + "RotDegPerCount";
   IF #OscHomeHighRelDeg > 360.0 THEN #OscHomeHighRelDeg := #OscHomeHighRelDeg - 360.0; END_IF;
   #OscHomeHigh2RelDeg := #OscHomeHighRelDeg + "RotDegPerCount";
   IF #OscHomeHigh2RelDeg > 360.0 THEN #OscHomeHigh2RelDeg := #OscHomeHigh2RelDeg - 360.0; END_IF;
   #OscHomeLowRelDeg := #OscHomeRelDeg - "RotDegPerCount";
   IF #OscHomeLowRelDeg < 0.0 THEN #OscHomeLowRelDeg := #OscHomeLowRelDeg - 360.0; END_IF;
   #OscHomeLow2RelDeg := #OscHomeLowRelDeg - "RotDegPerCount";
   IF #OscHomeLow2RelDeg < 0.0 THEN #OscHomeLow2RelDeg := #OscHomeLow2RelDeg - 360.0; END_IF;
END_REGION

REGION Network 13: Run Lamp Test
   // Turn on the lamp and horn test bits for the set amount of time and reset bit
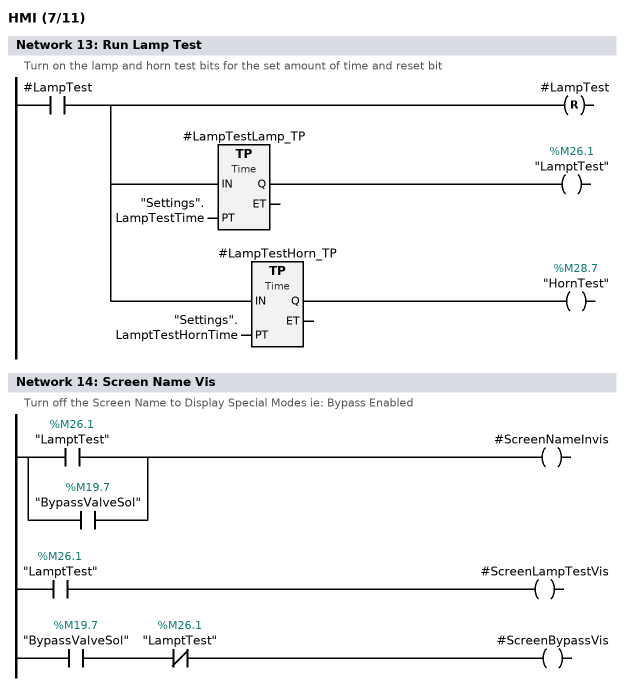
   RUNG wire#powerrail
      Contact( #LampTest )
      wire#w1
      R_Coil( #LampTest )
   END_RUNG
   RUNG wire#w1
      { S7_Templates := "time_type := Time" } #LampTestLamp_TP.TP(pt := "Settings".LampTestTime, et =>)
      Coil( "LamptTest" )
   END_RUNG
   RUNG wire#w1
      { S7_Templates := "time_type := Time" } #LampTestHorn_TP.TP(pt := "Settings".LamptTestHornTime, et =>)
      Coil( "HornTest" )
   END_RUNG
   // the same network as SCL:
   #_w1 := #LampTest;
   IF #_w1 THEN #LampTest := FALSE; END_IF;
   #LampTestLamp_TP(IN := #_w1, PT := "Settings".LampTestTime);   // TP
   "LamptTest" := #LampTestLamp_TP.Q;
   #LampTestHorn_TP(IN := #_w1, PT := "Settings".LamptTestHornTime);   // TP
   "HornTest" := #LampTestHorn_TP.Q;
END_REGION

REGION Network 14: Screen Name Vis
   // Turn off the Screen Name to Display Special Modes ie: Bypass Enabled
   RUNG wire#powerrail
      Contact( "LamptTest" )
      wire#w1
      Coil( #ScreenNameInvis )
   END_RUNG
   RUNG wire#powerrail
      Contact( "BypassValveSol" )
   END_RUNG wire#w1
   RUNG wire#powerrail
      Contact( "LamptTest" )
      Coil( #ScreenLampTestVis )
   END_RUNG
   RUNG wire#powerrail
      Contact( "BypassValveSol" )
      I_Contact( "LamptTest" )
      Coil( #ScreenBypassVis )
   END_RUNG
   // the same network as SCL:
   #ScreenNameInvis := "LamptTest" OR "BypassValveSol";
   #ScreenLampTestVis := "LamptTest";
   #ScreenBypassVis := "BypassValveSol" AND NOT "LamptTest";
END_REGION

